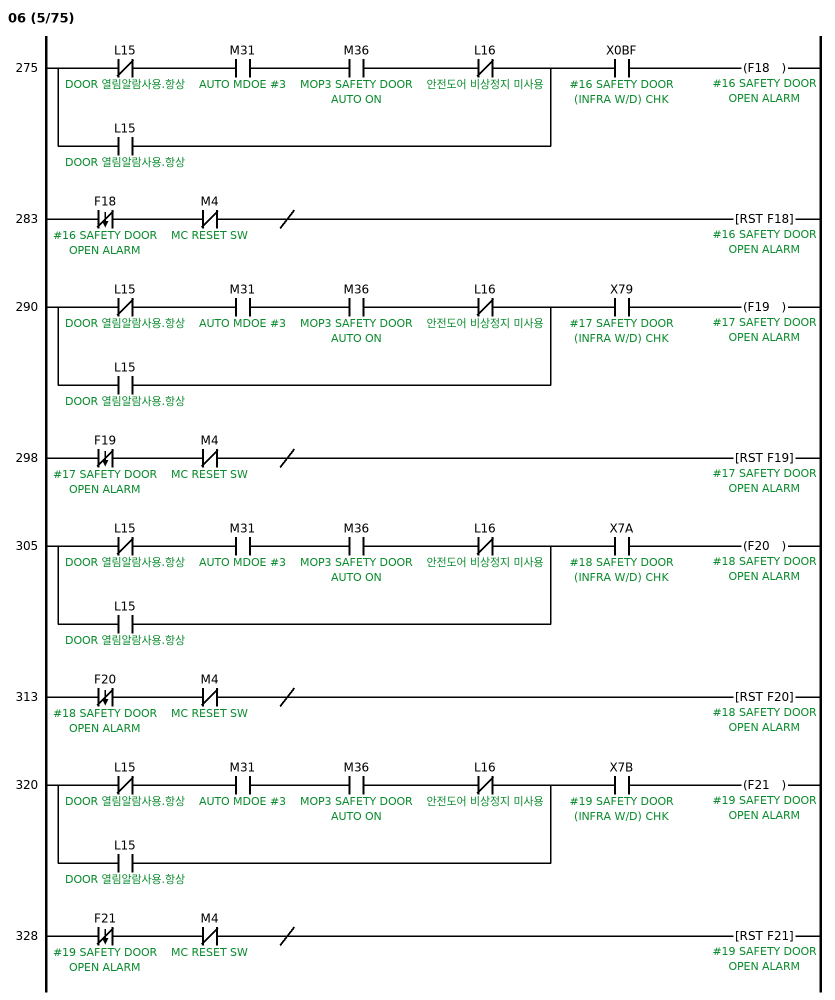
275   LDI     L15  ; DOOR 열림알람사용.항상
      AND     M31  ; AUTO MDOE #3
      AND     M36  ; MOP3 SAFETY DOOR AUTO ON
      ANI     L16  ; 안전도어 비상정지 미사용
      OR      L15  ; DOOR 열림알람사용.항상
      AND     X0BF  ; #16 SAFETY DOOR (INFRA W/D) CHK
      OUT     F18  ; #16 SAFETY DOOR OPEN ALARM
283   LDFI    F18  ; #16 SAFETY DOOR OPEN ALARM
      ANI     M4  ; MC RESET SW
      INV
      RST     F18  ; #16 SAFETY DOOR OPEN ALARM
290   LDI     L15  ; DOOR 열림알람사용.항상
      AND     M31  ; AUTO MDOE #3
      AND     M36  ; MOP3 SAFETY DOOR AUTO ON
      ANI     L16  ; 안전도어 비상정지 미사용
      OR      L15  ; DOOR 열림알람사용.항상
      AND     X79  ; #17 SAFETY DOOR (INFRA W/D) CHK
      OUT     F19  ; #17 SAFETY DOOR OPEN ALARM
298   LDFI    F19  ; #17 SAFETY DOOR OPEN ALARM
      ANI     M4  ; MC RESET SW
      INV
      RST     F19  ; #17 SAFETY DOOR OPEN ALARM
305   LDI     L15  ; DOOR 열림알람사용.항상
      AND     M31  ; AUTO MDOE #3
      AND     M36  ; MOP3 SAFETY DOOR AUTO ON
      ANI     L16  ; 안전도어 비상정지 미사용
      OR      L15  ; DOOR 열림알람사용.항상
      AND     X7A  ; #18 SAFETY DOOR (INFRA W/D) CHK
      OUT     F20  ; #18 SAFETY DOOR OPEN ALARM
313   LDFI    F20  ; #18 SAFETY DOOR OPEN ALARM
      ANI     M4  ; MC RESET SW
      INV
      RST     F20  ; #18 SAFETY DOOR OPEN ALARM
320   LDI     L15  ; DOOR 열림알람사용.항상
      AND     M31  ; AUTO MDOE #3
      AND     M36  ; MOP3 SAFETY DOOR AUTO ON
      ANI     L16  ; 안전도어 비상정지 미사용
      OR      L15  ; DOOR 열림알람사용.항상
      AND     X7B  ; #19 SAFETY DOOR (INFRA W/D) CHK
      OUT     F21  ; #19 SAFETY DOOR OPEN ALARM
328   LDFI    F21  ; #19 SAFETY DOOR OPEN ALARM
      ANI     M4  ; MC RESET SW
      INV
      RST     F21  ; #19 SAFETY DOOR OPEN ALARM
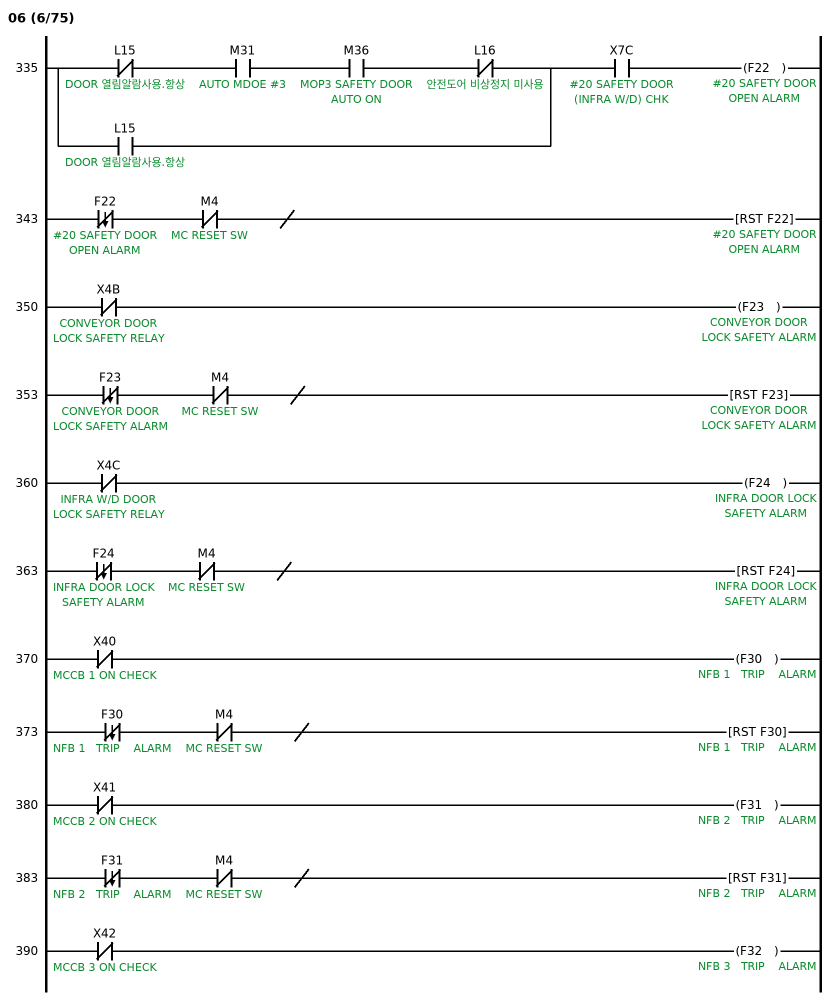
335   LDI     L15  ; DOOR 열림알람사용.항상
      AND     M31  ; AUTO MDOE #3
      AND     M36  ; MOP3 SAFETY DOOR AUTO ON
      ANI     L16  ; 안전도어 비상정지 미사용
      OR      L15  ; DOOR 열림알람사용.항상
      AND     X7C  ; #20 SAFETY DOOR (INFRA W/D) CHK
      OUT     F22  ; #20 SAFETY DOOR OPEN ALARM
343   LDFI    F22  ; #20 SAFETY DOOR OPEN ALARM
      ANI     M4  ; MC RESET SW
      INV
      RST     F22  ; #20 SAFETY DOOR OPEN ALARM
350   LDI     X4B  ; CONVEYOR DOOR LOCK SAFETY RELAY
      OUT     F23  ; CONVEYOR DOOR LOCK SAFETY ALARM
353   LDFI    F23  ; CONVEYOR DOOR LOCK SAFETY ALARM
      ANI     M4  ; MC RESET SW
      INV
      RST     F23  ; CONVEYOR DOOR LOCK SAFETY ALARM
360   LDI     X4C  ; INFRA W/D DOOR LOCK SAFETY RELAY
      OUT     F24  ; INFRA DOOR LOCK SAFETY ALARM
363   LDFI    F24  ; INFRA DOOR LOCK SAFETY ALARM
      ANI     M4  ; MC RESET SW
      INV
      RST     F24  ; INFRA DOOR LOCK SAFETY ALARM
370   LDI     X40  ; MCCB 1 ON CHECK
      OUT     F30  ; NFB 1   TRIP    ALARM
373   LDFI    F30  ; NFB 1   TRIP    ALARM
      ANI     M4  ; MC RESET SW
      INV
      RST     F30  ; NFB 1   TRIP    ALARM
380   LDI     X41  ; MCCB 2 ON CHECK
      OUT     F31  ; NFB 2   TRIP    ALARM
383   LDFI    F31  ; NFB 2   TRIP    ALARM
      ANI     M4  ; MC RESET SW
      INV
      RST     F31  ; NFB 2   TRIP    ALARM
390   LDI     X42  ; MCCB 3 ON CHECK
      OUT     F32  ; NFB 3   TRIP    ALARM
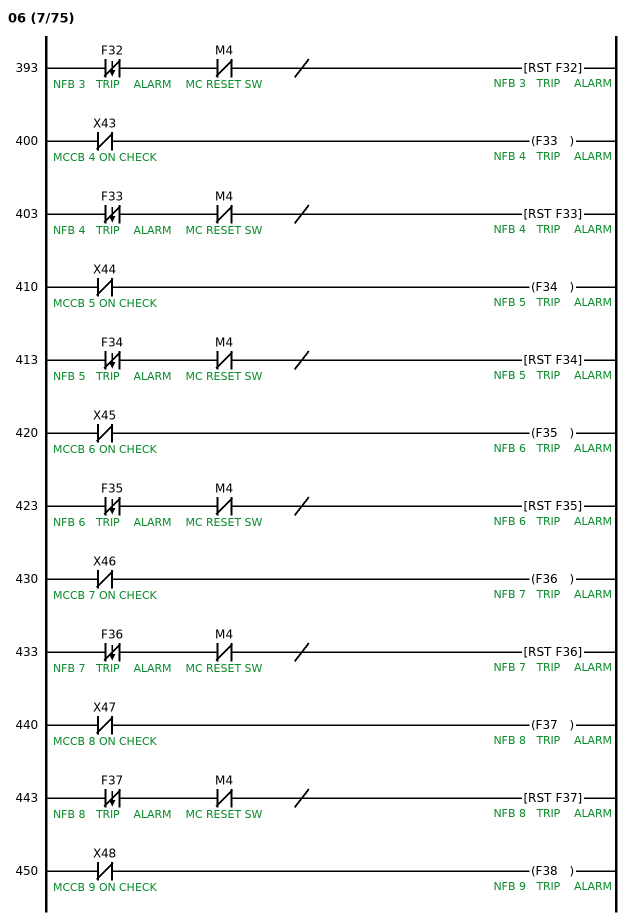
393   LDFI    F32  ; NFB 3   TRIP    ALARM
      ANI     M4  ; MC RESET SW
      INV
      RST     F32  ; NFB 3   TRIP    ALARM
400   LDI     X43  ; MCCB 4 ON CHECK
      OUT     F33  ; NFB 4   TRIP    ALARM
403   LDFI    F33  ; NFB 4   TRIP    ALARM
      ANI     M4  ; MC RESET SW
      INV
      RST     F33  ; NFB 4   TRIP    ALARM
410   LDI     X44  ; MCCB 5 ON CHECK
      OUT     F34  ; NFB 5   TRIP    ALARM
413   LDFI    F34  ; NFB 5   TRIP    ALARM
      ANI     M4  ; MC RESET SW
      INV
      RST     F34  ; NFB 5   TRIP    ALARM
420   LDI     X45  ; MCCB 6 ON CHECK
      OUT     F35  ; NFB 6   TRIP    ALARM
423   LDFI    F35  ; NFB 6   TRIP    ALARM
      ANI     M4  ; MC RESET SW
      INV
      RST     F35  ; NFB 6   TRIP    ALARM
430   LDI     X46  ; MCCB 7 ON CHECK
      OUT     F36  ; NFB 7   TRIP    ALARM
433   LDFI    F36  ; NFB 7   TRIP    ALARM
      ANI     M4  ; MC RESET SW
      INV
      RST     F36  ; NFB 7   TRIP    ALARM
440   LDI     X47  ; MCCB 8 ON CHECK
      OUT     F37  ; NFB 8   TRIP    ALARM
443   LDFI    F37  ; NFB 8   TRIP    ALARM
      ANI     M4  ; MC RESET SW
      INV
      RST     F37  ; NFB 8   TRIP    ALARM
450   LDI     X48  ; MCCB 9 ON CHECK
      OUT     F38  ; NFB 9   TRIP    ALARM
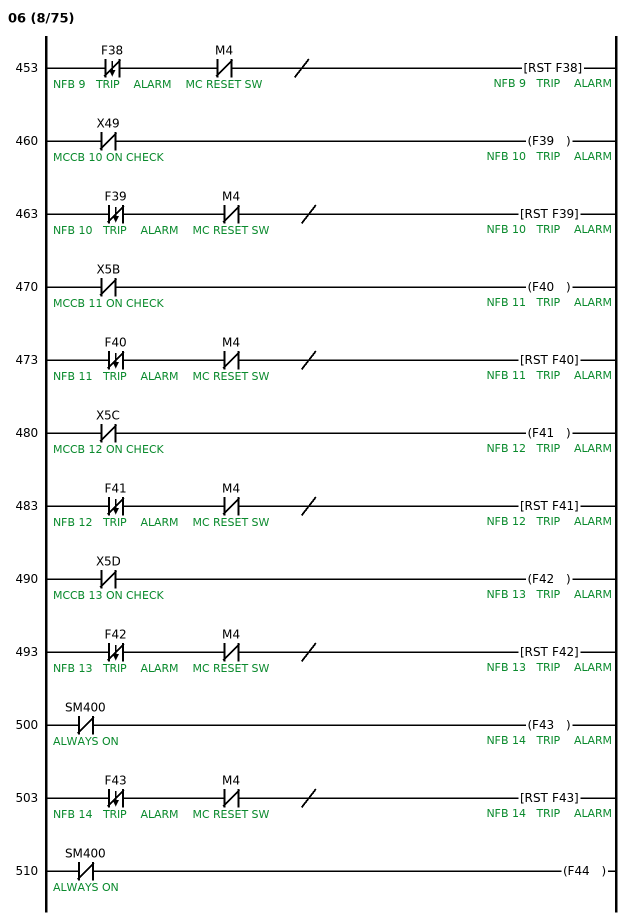
453   LDFI    F38  ; NFB 9   TRIP    ALARM
      ANI     M4  ; MC RESET SW
      INV
      RST     F38  ; NFB 9   TRIP    ALARM
460   LDI     X49  ; MCCB 10 ON CHECK
      OUT     F39  ; NFB 10   TRIP    ALARM
463   LDFI    F39  ; NFB 10   TRIP    ALARM
      ANI     M4  ; MC RESET SW
      INV
      RST     F39  ; NFB 10   TRIP    ALARM
470   LDI     X5B  ; MCCB 11 ON CHECK
      OUT     F40  ; NFB 11   TRIP    ALARM
473   LDFI    F40  ; NFB 11   TRIP    ALARM
      ANI     M4  ; MC RESET SW
      INV
      RST     F40  ; NFB 11   TRIP    ALARM
480   LDI     X5C  ; MCCB 12 ON CHECK
      OUT     F41  ; NFB 12   TRIP    ALARM
483   LDFI    F41  ; NFB 12   TRIP    ALARM
      ANI     M4  ; MC RESET SW
      INV
      RST     F41  ; NFB 12   TRIP    ALARM
490   LDI     X5D  ; MCCB 13 ON CHECK
      OUT     F42  ; NFB 13   TRIP    ALARM
493   LDFI    F42  ; NFB 13   TRIP    ALARM
      ANI     M4  ; MC RESET SW
      INV
      RST     F42  ; NFB 13   TRIP    ALARM
500   LDI     SM400  ; ALWAYS ON
      OUT     F43  ; NFB 14   TRIP    ALARM
503   LDFI    F43  ; NFB 14   TRIP    ALARM
      ANI     M4  ; MC RESET SW
      INV
      RST     F43  ; NFB 14   TRIP    ALARM
510   LDI     SM400  ; ALWAYS ON
      OUT     F44
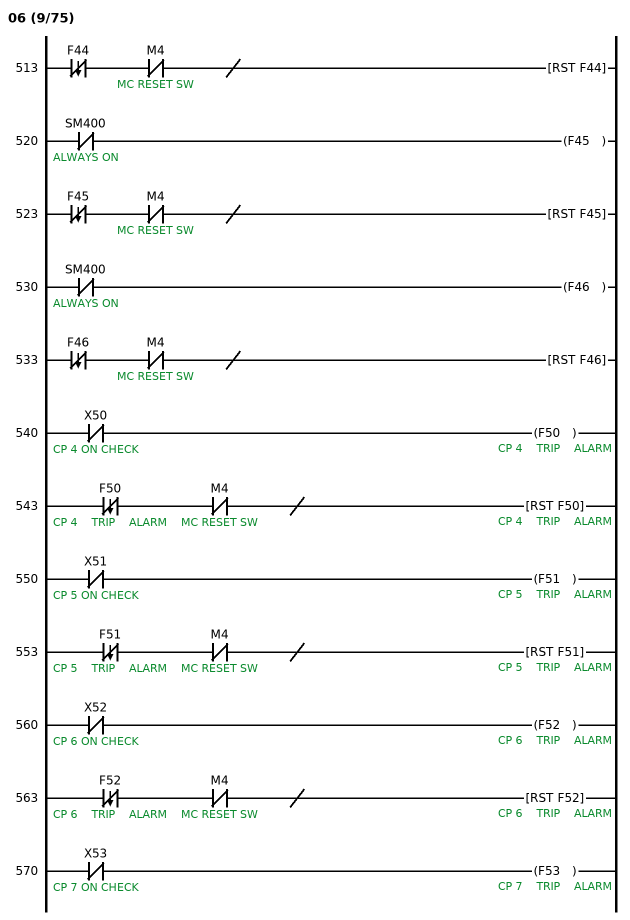
513   LDFI    F44
      ANI     M4  ; MC RESET SW
      INV
      RST     F44
520   LDI     SM400  ; ALWAYS ON
      OUT     F45
523   LDFI    F45
      ANI     M4  ; MC RESET SW
      INV
      RST     F45
530   LDI     SM400  ; ALWAYS ON
      OUT     F46
533   LDFI    F46
      ANI     M4  ; MC RESET SW
      INV
      RST     F46
540   LDI     X50  ; CP 4 ON CHECK
      OUT     F50  ; CP 4    TRIP    ALARM
543   LDFI    F50  ; CP 4    TRIP    ALARM
      ANI     M4  ; MC RESET SW
      INV
      RST     F50  ; CP 4    TRIP    ALARM
550   LDI     X51  ; CP 5 ON CHECK
      OUT     F51  ; CP 5    TRIP    ALARM
553   LDFI    F51  ; CP 5    TRIP    ALARM
      ANI     M4  ; MC RESET SW
      INV
      RST     F51  ; CP 5    TRIP    ALARM
560   LDI     X52  ; CP 6 ON CHECK
      OUT     F52  ; CP 6    TRIP    ALARM
563   LDFI    F52  ; CP 6    TRIP    ALARM
      ANI     M4  ; MC RESET SW
      INV
      RST     F52  ; CP 6    TRIP    ALARM
570   LDI     X53  ; CP 7 ON CHECK
      OUT     F53  ; CP 7    TRIP    ALARM
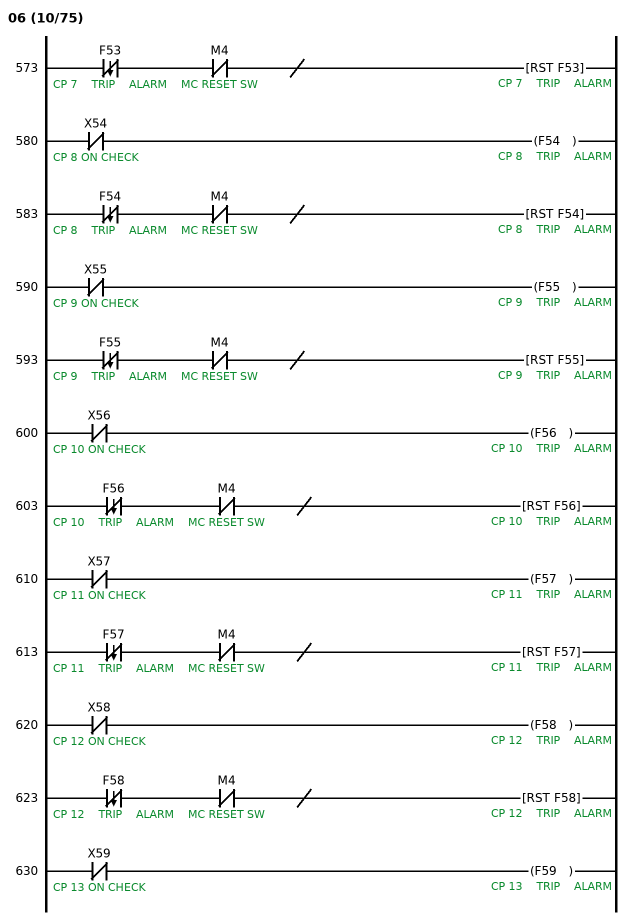
573   LDFI    F53  ; CP 7    TRIP    ALARM
      ANI     M4  ; MC RESET SW
      INV
      RST     F53  ; CP 7    TRIP    ALARM
580   LDI     X54  ; CP 8 ON CHECK
      OUT     F54  ; CP 8    TRIP    ALARM
583   LDFI    F54  ; CP 8    TRIP    ALARM
      ANI     M4  ; MC RESET SW
      INV
      RST     F54  ; CP 8    TRIP    ALARM
590   LDI     X55  ; CP 9 ON CHECK
      OUT     F55  ; CP 9    TRIP    ALARM
593   LDFI    F55  ; CP 9    TRIP    ALARM
      ANI     M4  ; MC RESET SW
      INV
      RST     F55  ; CP 9    TRIP    ALARM
600   LDI     X56  ; CP 10 ON CHECK
      OUT     F56  ; CP 10    TRIP    ALARM
603   LDFI    F56  ; CP 10    TRIP    ALARM
      ANI     M4  ; MC RESET SW
      INV
      RST     F56  ; CP 10    TRIP    ALARM
610   LDI     X57  ; CP 11 ON CHECK
      OUT     F57  ; CP 11    TRIP    ALARM
613   LDFI    F57  ; CP 11    TRIP    ALARM
      ANI     M4  ; MC RESET SW
      INV
      RST     F57  ; CP 11    TRIP    ALARM
620   LDI     X58  ; CP 12 ON CHECK
      OUT     F58  ; CP 12    TRIP    ALARM
623   LDFI    F58  ; CP 12    TRIP    ALARM
      ANI     M4  ; MC RESET SW
      INV
      RST     F58  ; CP 12    TRIP    ALARM
630   LDI     X59  ; CP 13 ON CHECK
      OUT     F59  ; CP 13    TRIP    ALARM
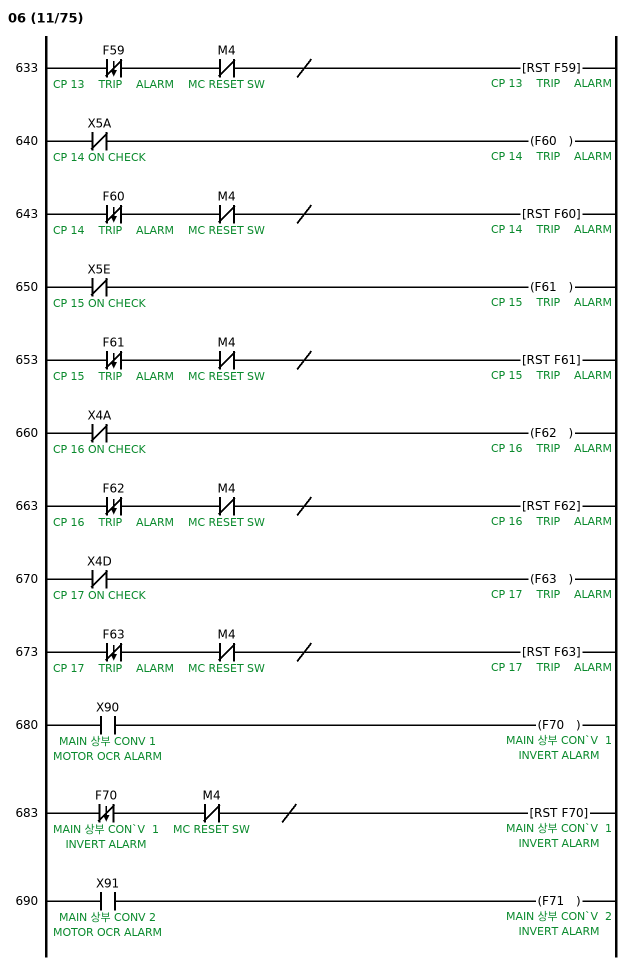
633   LDFI    F59  ; CP 13    TRIP    ALARM
      ANI     M4  ; MC RESET SW
      INV
      RST     F59  ; CP 13    TRIP    ALARM
640   LDI     X5A  ; CP 14 ON CHECK
      OUT     F60  ; CP 14    TRIP    ALARM
643   LDFI    F60  ; CP 14    TRIP    ALARM
      ANI     M4  ; MC RESET SW
      INV
      RST     F60  ; CP 14    TRIP    ALARM
650   LDI     X5E  ; CP 15 ON CHECK
      OUT     F61  ; CP 15    TRIP    ALARM
653   LDFI    F61  ; CP 15    TRIP    ALARM
      ANI     M4  ; MC RESET SW
      INV
      RST     F61  ; CP 15    TRIP    ALARM
660   LDI     X4A  ; CP 16 ON CHECK
      OUT     F62  ; CP 16    TRIP    ALARM
663   LDFI    F62  ; CP 16    TRIP    ALARM
      ANI     M4  ; MC RESET SW
      INV
      RST     F62  ; CP 16    TRIP    ALARM
670   LDI     X4D  ; CP 17 ON CHECK
      OUT     F63  ; CP 17    TRIP    ALARM
673   LDFI    F63  ; CP 17    TRIP    ALARM
      ANI     M4  ; MC RESET SW
      INV
      RST     F63  ; CP 17    TRIP    ALARM
680   LD      X90  ; MAIN 상부 CONV 1 MOTOR OCR ALARM
      OUT     F70  ; MAIN 상부 CON`V  1 INVERT ALARM
683   LDFI    F70  ; MAIN 상부 CON`V  1 INVERT ALARM
      ANI     M4  ; MC RESET SW
      INV
      RST     F70  ; MAIN 상부 CON`V  1 INVERT ALARM
690   LD      X91  ; MAIN 상부 CONV 2 MOTOR OCR ALARM
      OUT     F71  ; MAIN 상부 CON`V  2 INVERT ALARM
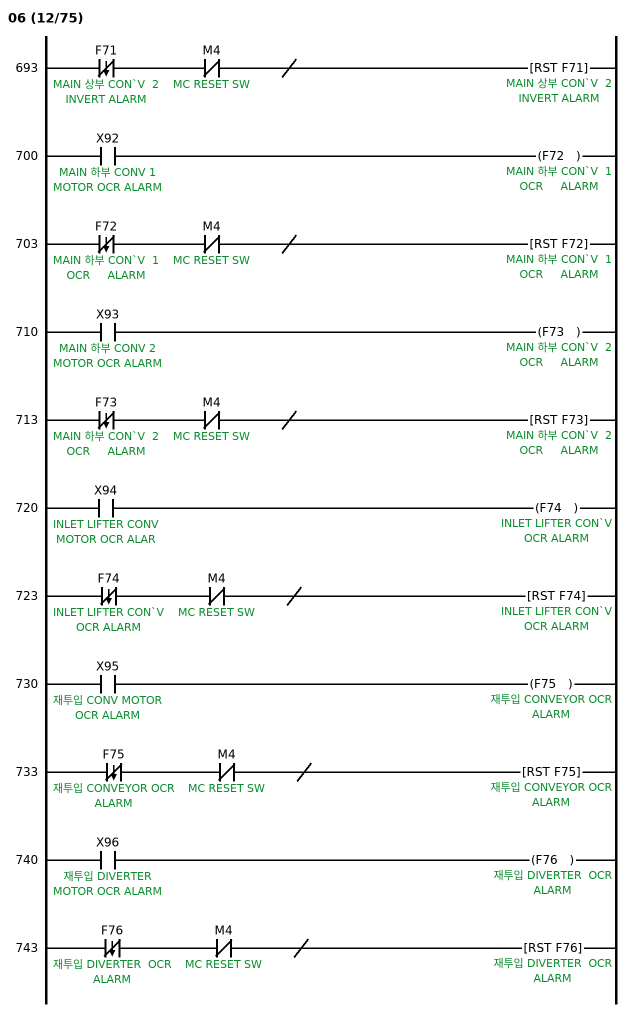
693   LDFI    F71  ; MAIN 상부 CON`V  2 INVERT ALARM
      ANI     M4  ; MC RESET SW
      INV
      RST     F71  ; MAIN 상부 CON`V  2 INVERT ALARM
700   LD      X92  ; MAIN 하부 CONV 1 MOTOR OCR ALARM
      OUT     F72  ; MAIN 하부 CON`V  1 OCR     ALARM
703   LDFI    F72  ; MAIN 하부 CON`V  1 OCR     ALARM
      ANI     M4  ; MC RESET SW
      INV
      RST     F72  ; MAIN 하부 CON`V  1 OCR     ALARM
710   LD      X93  ; MAIN 하부 CONV 2 MOTOR OCR ALARM
      OUT     F73  ; MAIN 하부 CON`V  2 OCR     ALARM
713   LDFI    F73  ; MAIN 하부 CON`V  2 OCR     ALARM
      ANI     M4  ; MC RESET SW
      INV
      RST     F73  ; MAIN 하부 CON`V  2 OCR     ALARM
720   LD      X94  ; INLET LIFTER CONV MOTOR OCR ALAR
      OUT     F74  ; INLET LIFTER CON`V OCR ALARM
723   LDFI    F74  ; INLET LIFTER CON`V OCR ALARM
      ANI     M4  ; MC RESET SW
      INV
      RST     F74  ; INLET LIFTER CON`V OCR ALARM
730   LD      X95  ; 재투입 CONV MOTOR OCR ALARM
      OUT     F75  ; 재투입 CONVEYOR OCR     ALARM
733   LDFI    F75  ; 재투입 CONVEYOR OCR     ALARM
      ANI     M4  ; MC RESET SW
      INV
      RST     F75  ; 재투입 CONVEYOR OCR     ALARM
740   LD      X96  ; 재투입 DIVERTER MOTOR OCR ALARM
      OUT     F76  ; 재투입 DIVERTER  OCR     ALARM
743   LDFI    F76  ; 재투입 DIVERTER  OCR     ALARM
      ANI     M4  ; MC RESET SW
      INV
      RST     F76  ; 재투입 DIVERTER  OCR     ALARM
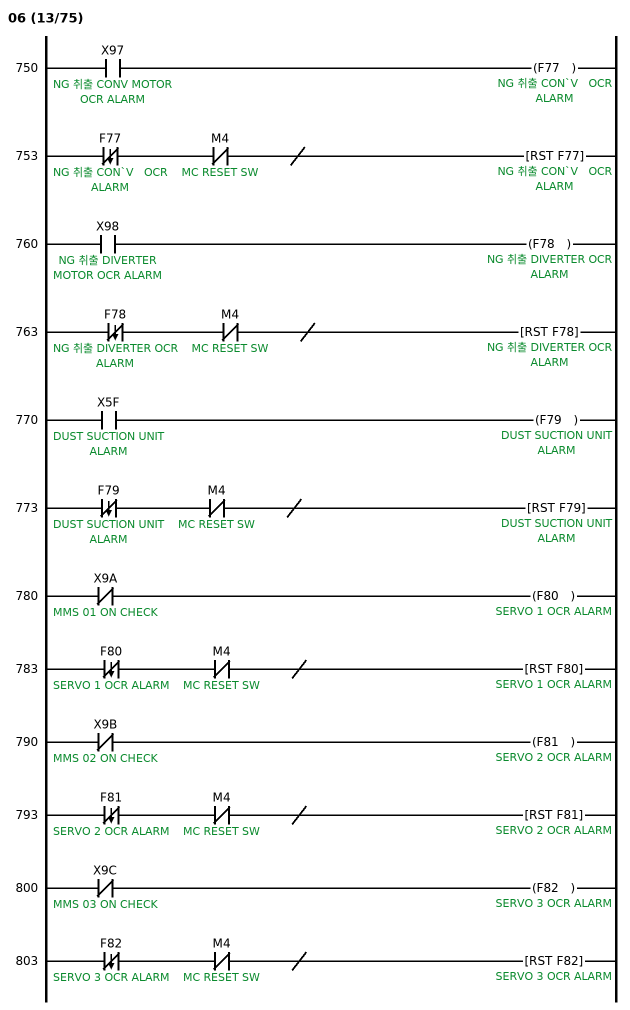
750   LD      X97  ; NG 취출 CONV MOTOR OCR ALARM
      OUT     F77  ; NG 취출 CON`V   OCR     ALARM
753   LDFI    F77  ; NG 취출 CON`V   OCR     ALARM
      ANI     M4  ; MC RESET SW
      INV
      RST     F77  ; NG 취출 CON`V   OCR     ALARM
760   LD      X98  ; NG 취출 DIVERTER MOTOR OCR ALARM
      OUT     F78  ; NG 취출 DIVERTER OCR ALARM
763   LDFI    F78  ; NG 취출 DIVERTER OCR ALARM
      ANI     M4  ; MC RESET SW
      INV
      RST     F78  ; NG 취출 DIVERTER OCR ALARM
770   LD      X5F  ; DUST SUCTION UNIT ALARM
      OUT     F79  ; DUST SUCTION UNIT ALARM
773   LDFI    F79  ; DUST SUCTION UNIT ALARM
      ANI     M4  ; MC RESET SW
      INV
      RST     F79  ; DUST SUCTION UNIT ALARM
780   LDI     X9A  ; MMS 01 ON CHECK
      OUT     F80  ; SERVO 1 OCR ALARM
783   LDFI    F80  ; SERVO 1 OCR ALARM
      ANI     M4  ; MC RESET SW
      INV
      RST     F80  ; SERVO 1 OCR ALARM
790   LDI     X9B  ; MMS 02 ON CHECK
      OUT     F81  ; SERVO 2 OCR ALARM
793   LDFI    F81  ; SERVO 2 OCR ALARM
      ANI     M4  ; MC RESET SW
      INV
      RST     F81  ; SERVO 2 OCR ALARM
800   LDI     X9C  ; MMS 03 ON CHECK
      OUT     F82  ; SERVO 3 OCR ALARM
803   LDFI    F82  ; SERVO 3 OCR ALARM
      ANI     M4  ; MC RESET SW
      INV
      RST     F82  ; SERVO 3 OCR ALARM
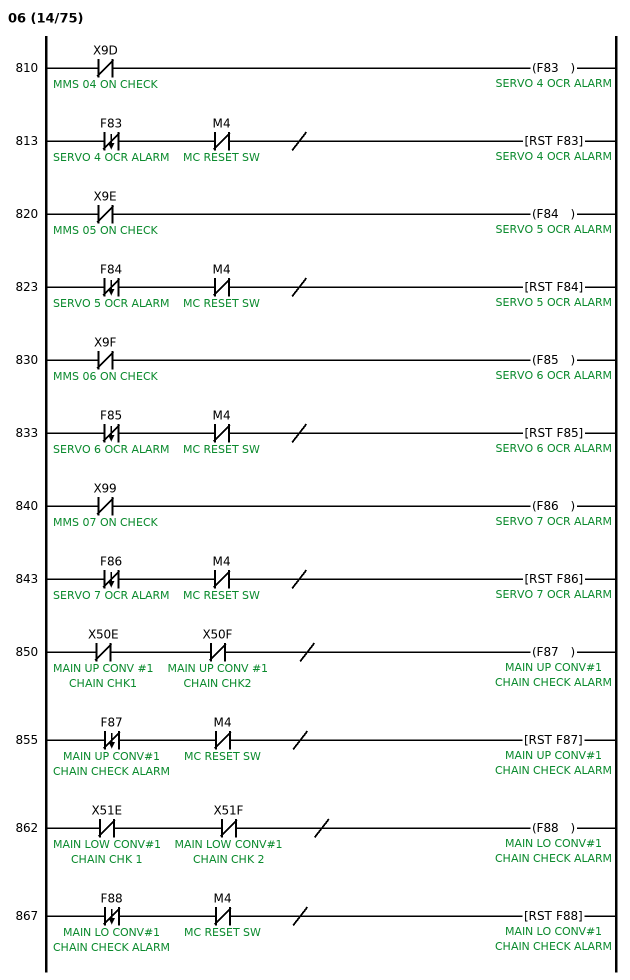
810   LDI     X9D  ; MMS 04 ON CHECK
      OUT     F83  ; SERVO 4 OCR ALARM
813   LDFI    F83  ; SERVO 4 OCR ALARM
      ANI     M4  ; MC RESET SW
      INV
      RST     F83  ; SERVO 4 OCR ALARM
820   LDI     X9E  ; MMS 05 ON CHECK
      OUT     F84  ; SERVO 5 OCR ALARM
823   LDFI    F84  ; SERVO 5 OCR ALARM
      ANI     M4  ; MC RESET SW
      INV
      RST     F84  ; SERVO 5 OCR ALARM
830   LDI     X9F  ; MMS 06 ON CHECK
      OUT     F85  ; SERVO 6 OCR ALARM
833   LDFI    F85  ; SERVO 6 OCR ALARM
      ANI     M4  ; MC RESET SW
      INV
      RST     F85  ; SERVO 6 OCR ALARM
840   LDI     X99  ; MMS 07 ON CHECK
      OUT     F86  ; SERVO 7 OCR ALARM
843   LDFI    F86  ; SERVO 7 OCR ALARM
      ANI     M4  ; MC RESET SW
      INV
      RST     F86  ; SERVO 7 OCR ALARM
850   LDI     X50E  ; MAIN UP CONV #1 CHAIN CHK1
      ANI     X50F  ; MAIN UP CONV #1 CHAIN CHK2
      INV
      OUT     F87  ; MAIN UP CONV#1 CHAIN CHECK ALARM
855   LDFI    F87  ; MAIN UP CONV#1 CHAIN CHECK ALARM
      ANI     M4  ; MC RESET SW
      INV
      RST     F87  ; MAIN UP CONV#1 CHAIN CHECK ALARM
862   LDI     X51E  ; MAIN LOW CONV#1 CHAIN CHK 1
      ANI     X51F  ; MAIN LOW CONV#1 CHAIN CHK 2
      INV
      OUT     F88  ; MAIN LO CONV#1 CHAIN CHECK ALARM
867   LDFI    F88  ; MAIN LO CONV#1 CHAIN CHECK ALARM
      ANI     M4  ; MC RESET SW
      INV
      RST     F88  ; MAIN LO CONV#1 CHAIN CHECK ALARM
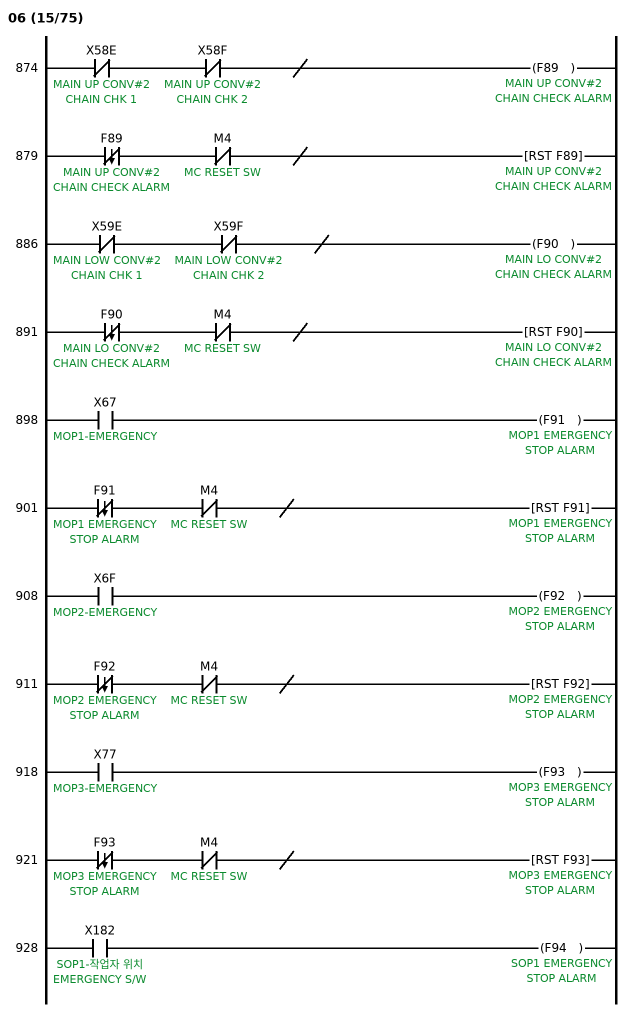
874   LDI     X58E  ; MAIN UP CONV#2 CHAIN CHK 1
      ANI     X58F  ; MAIN UP CONV#2 CHAIN CHK 2
      INV
      OUT     F89  ; MAIN UP CONV#2 CHAIN CHECK ALARM
879   LDFI    F89  ; MAIN UP CONV#2 CHAIN CHECK ALARM
      ANI     M4  ; MC RESET SW
      INV
      RST     F89  ; MAIN UP CONV#2 CHAIN CHECK ALARM
886   LDI     X59E  ; MAIN LOW CONV#2 CHAIN CHK 1
      ANI     X59F  ; MAIN LOW CONV#2 CHAIN CHK 2
      INV
      OUT     F90  ; MAIN LO CONV#2 CHAIN CHECK ALARM
891   LDFI    F90  ; MAIN LO CONV#2 CHAIN CHECK ALARM
      ANI     M4  ; MC RESET SW
      INV
      RST     F90  ; MAIN LO CONV#2 CHAIN CHECK ALARM
898   LD      X67  ; MOP1-EMERGENCY
      OUT     F91  ; MOP1 EMERGENCY STOP ALARM
901   LDFI    F91  ; MOP1 EMERGENCY STOP ALARM
      ANI     M4  ; MC RESET SW
      INV
      RST     F91  ; MOP1 EMERGENCY STOP ALARM
908   LD      X6F  ; MOP2-EMERGENCY
      OUT     F92  ; MOP2 EMERGENCY STOP ALARM
911   LDFI    F92  ; MOP2 EMERGENCY STOP ALARM
      ANI     M4  ; MC RESET SW
      INV
      RST     F92  ; MOP2 EMERGENCY STOP ALARM
918   LD      X77  ; MOP3-EMERGENCY
      OUT     F93  ; MOP3 EMERGENCY STOP ALARM
921   LDFI    F93  ; MOP3 EMERGENCY STOP ALARM
      ANI     M4  ; MC RESET SW
      INV
      RST     F93  ; MOP3 EMERGENCY STOP ALARM
928   LD      X182  ; SOP1-작업자 위치 EMERGENCY S/W
      OUT     F94  ; SOP1 EMERGENCY STOP ALARM
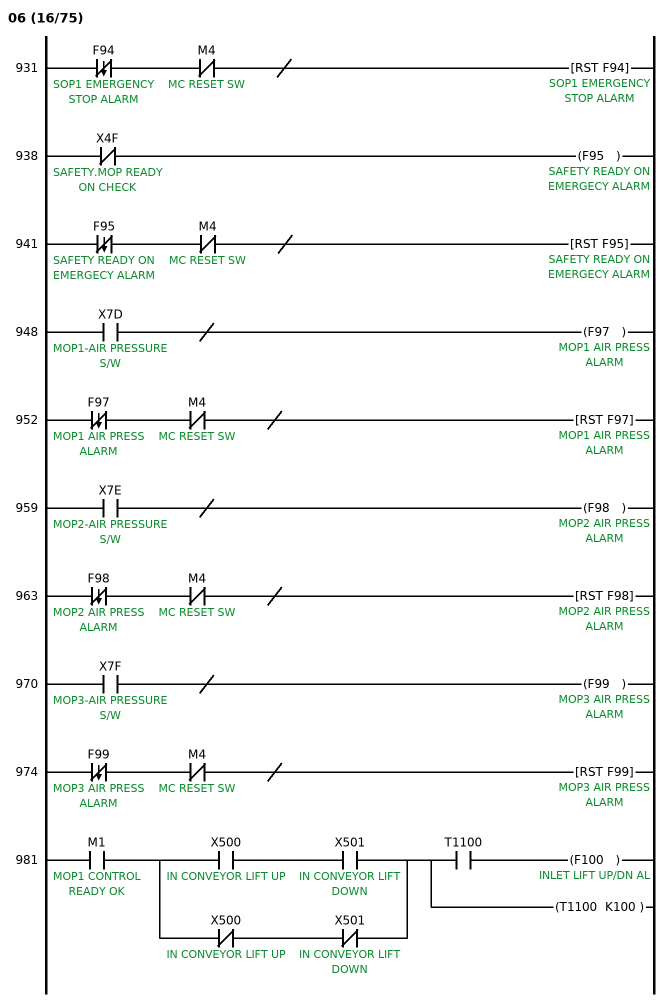
931   LDFI    F94  ; SOP1 EMERGENCY STOP ALARM
      ANI     M4  ; MC RESET SW
      INV
      RST     F94  ; SOP1 EMERGENCY STOP ALARM
938   LDI     X4F  ; SAFETY.MOP READY ON CHECK
      OUT     F95  ; SAFETY READY ON EMERGECY ALARM
941   LDFI    F95  ; SAFETY READY ON EMERGECY ALARM
      ANI     M4  ; MC RESET SW
      INV
      RST     F95  ; SAFETY READY ON EMERGECY ALARM
948   LD      X7D  ; MOP1-AIR PRESSURE S/W
      INV
      OUT     F97  ; MOP1 AIR PRESS ALARM
952   LDFI    F97  ; MOP1 AIR PRESS ALARM
      ANI     M4  ; MC RESET SW
      INV
      RST     F97  ; MOP1 AIR PRESS ALARM
959   LD      X7E  ; MOP2-AIR PRESSURE S/W
      INV
      OUT     F98  ; MOP2 AIR PRESS ALARM
963   LDFI    F98  ; MOP2 AIR PRESS ALARM
      ANI     M4  ; MC RESET SW
      INV
      RST     F98  ; MOP2 AIR PRESS ALARM
970   LD      X7F  ; MOP3-AIR PRESSURE S/W
      INV
      OUT     F99  ; MOP3 AIR PRESS ALARM
974   LDFI    F99  ; MOP3 AIR PRESS ALARM
      ANI     M4  ; MC RESET SW
      INV
      RST     F99  ; MOP3 AIR PRESS ALARM
981   LD      M1  ; MOP1 CONTROL READY OK
      LD      X500  ; IN CONVEYOR LIFT UP
      AND     X501  ; IN CONVEYOR LIFT DOWN
      LDI     X500  ; IN CONVEYOR LIFT UP
      ANI     X501  ; IN CONVEYOR LIFT DOWN
      ORB
      ANB
      MPS
      AND     T1100
      OUT     F100  ; INLET LIFT UP/DN AL
      MPP
      OUT     T1100 K100
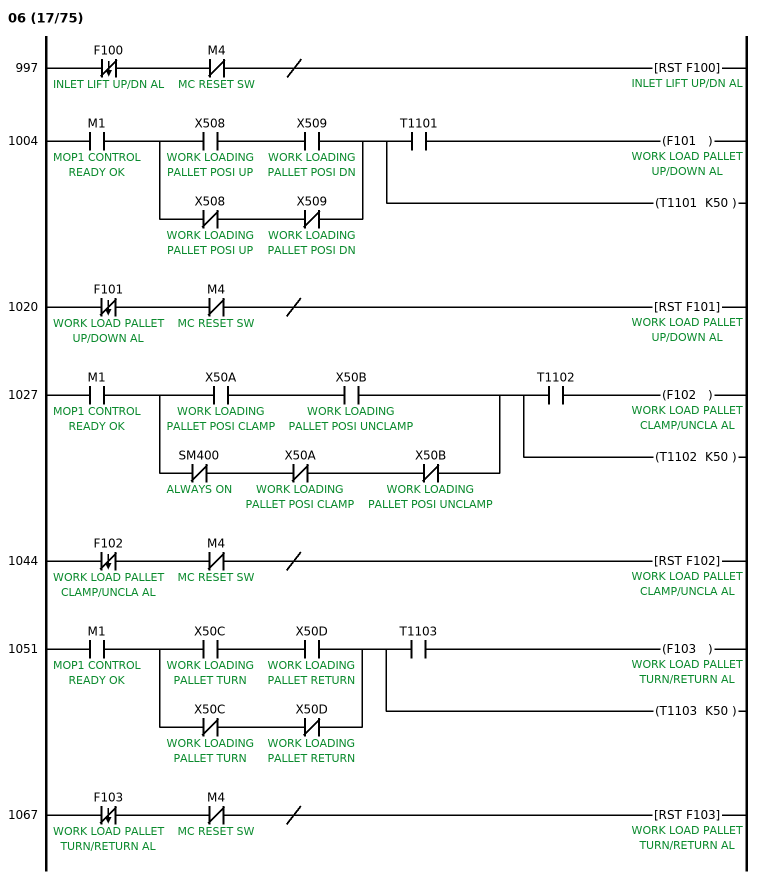
997   LDFI    F100  ; INLET LIFT UP/DN AL
      ANI     M4  ; MC RESET SW
      INV
      RST     F100  ; INLET LIFT UP/DN AL
1004  LD      M1  ; MOP1 CONTROL READY OK
      LD      X508  ; WORK LOADING PALLET POSI UP
      AND     X509  ; WORK LOADING PALLET POSI DN
      LDI     X508  ; WORK LOADING PALLET POSI UP
      ANI     X509  ; WORK LOADING PALLET POSI DN
      ORB
      ANB
      MPS
      AND     T1101
      OUT     F101  ; WORK LOAD PALLET UP/DOWN AL
      MPP
      OUT     T1101 K50
1020  LDFI    F101  ; WORK LOAD PALLET UP/DOWN AL
      ANI     M4  ; MC RESET SW
      INV
      RST     F101  ; WORK LOAD PALLET UP/DOWN AL
1027  LD      M1  ; MOP1 CONTROL READY OK
      LD      X50A  ; WORK LOADING PALLET POSI CLAMP
      AND     X50B  ; WORK LOADING PALLET POSI UNCLAMP
      LDI     SM400  ; ALWAYS ON
      ANI     X50A  ; WORK LOADING PALLET POSI CLAMP
      ANI     X50B  ; WORK LOADING PALLET POSI UNCLAMP
      ORB
      ANB
      MPS
      AND     T1102
      OUT     F102  ; WORK LOAD PALLET CLAMP/UNCLA AL
      MPP
      OUT     T1102 K50
1044  LDFI    F102  ; WORK LOAD PALLET CLAMP/UNCLA AL
      ANI     M4  ; MC RESET SW
      INV
      RST     F102  ; WORK LOAD PALLET CLAMP/UNCLA AL
1051  LD      M1  ; MOP1 CONTROL READY OK
      LD      X50C  ; WORK LOADING PALLET TURN
      AND     X50D  ; WORK LOADING PALLET RETURN
      LDI     X50C  ; WORK LOADING PALLET TURN
      ANI     X50D  ; WORK LOADING PALLET RETURN
      ORB
      ANB
      MPS
      AND     T1103
      OUT     F103  ; WORK LOAD PALLET TURN/RETURN AL
      MPP
      OUT     T1103 K50
1067  LDFI    F103  ; WORK LOAD PALLET TURN/RETURN AL
      ANI     M4  ; MC RESET SW
      INV
      RST     F103  ; WORK LOAD PALLET TURN/RETURN AL
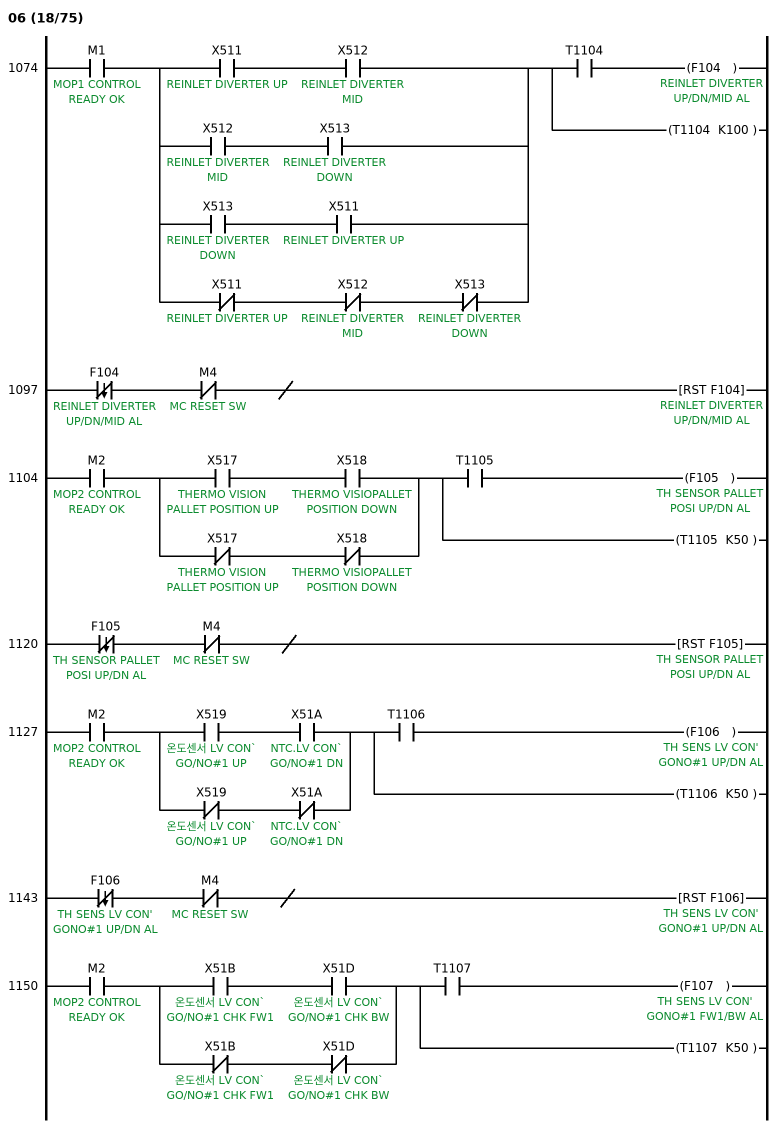
1074  LD      M1  ; MOP1 CONTROL READY OK
      LD      X511  ; REINLET DIVERTER UP
      AND     X512  ; REINLET DIVERTER MID
      LD      X512  ; REINLET DIVERTER MID
      AND     X513  ; REINLET DIVERTER DOWN
      ORB
      LD      X513  ; REINLET DIVERTER DOWN
      AND     X511  ; REINLET DIVERTER UP
      ORB
      LDI     X511  ; REINLET DIVERTER UP
      ANI     X512  ; REINLET DIVERTER MID
      ANI     X513  ; REINLET DIVERTER DOWN
      ORB
      ANB
      MPS
      AND     T1104
      OUT     F104  ; REINLET DIVERTER UP/DN/MID AL
      MPP
      OUT     T1104 K100
1097  LDFI    F104  ; REINLET DIVERTER UP/DN/MID AL
      ANI     M4  ; MC RESET SW
      INV
      RST     F104  ; REINLET DIVERTER UP/DN/MID AL
1104  LD      M2  ; MOP2 CONTROL READY OK
      LD      X517  ; THERMO VISION PALLET POSITION UP
      AND     X518  ; THERMO VISIOPALLET POSITION DOWN
      LDI     X517  ; THERMO VISION PALLET POSITION UP
      ANI     X518  ; THERMO VISIOPALLET POSITION DOWN
      ORB
      ANB
      MPS
      AND     T1105
      OUT     F105  ; TH SENSOR PALLET POSI UP/DN AL
      MPP
      OUT     T1105 K50
1120  LDFI    F105  ; TH SENSOR PALLET POSI UP/DN AL
      ANI     M4  ; MC RESET SW
      INV
      RST     F105  ; TH SENSOR PALLET POSI UP/DN AL
1127  LD      M2  ; MOP2 CONTROL READY OK
      LD      X519  ; 온도센서 LV CON` GO/NO#1 UP
      AND     X51A  ; NTC.LV CON` GO/NO#1 DN
      LDI     X519  ; 온도센서 LV CON` GO/NO#1 UP
      ANI     X51A  ; NTC.LV CON` GO/NO#1 DN
      ORB
      ANB
      MPS
      AND     T1106
      OUT     F106  ; TH SENS LV CON' GONO#1 UP/DN AL
      MPP
      OUT     T1106 K50
1143  LDFI    F106  ; TH SENS LV CON' GONO#1 UP/DN AL
      ANI     M4  ; MC RESET SW
      INV
      RST     F106  ; TH SENS LV CON' GONO#1 UP/DN AL
1150  LD      M2  ; MOP2 CONTROL READY OK
      LD      X51B  ; 온도센서 LV CON` GO/NO#1 CHK FW1
      AND     X51D  ; 온도센서 LV CON` GO/NO#1 CHK BW
      LDI     X51B  ; 온도센서 LV CON` GO/NO#1 CHK FW1
      ANI     X51D  ; 온도센서 LV CON` GO/NO#1 CHK BW
      ORB
      ANB
      MPS
      AND     T1107
      OUT     F107  ; TH SENS LV CON' GONO#1 FW1/BW AL
      MPP
      OUT     T1107 K50
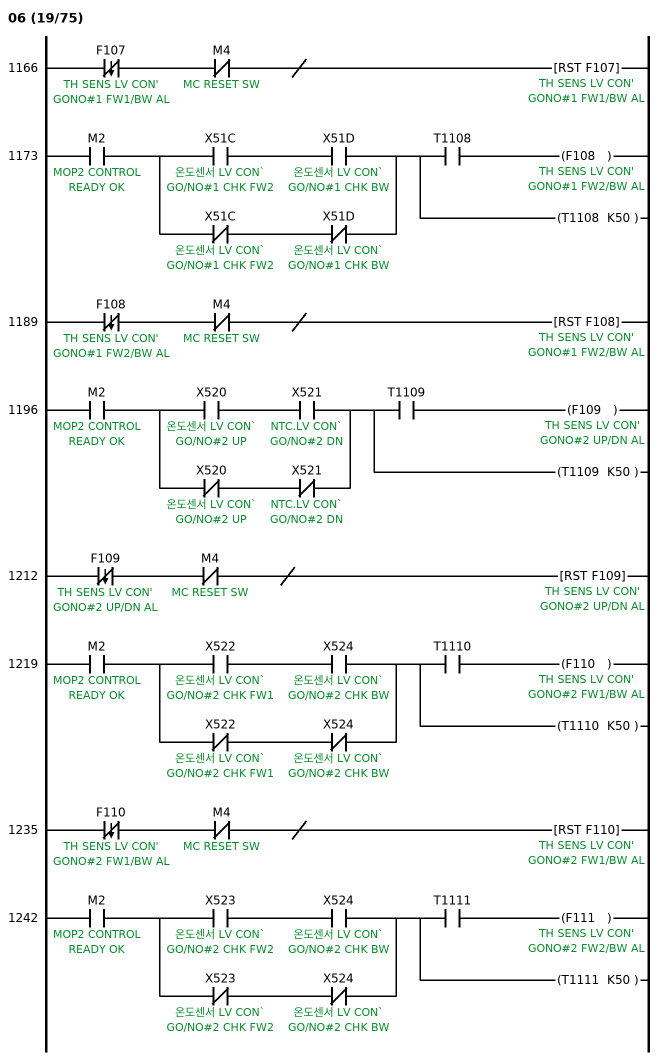
1166  LDFI    F107  ; TH SENS LV CON' GONO#1 FW1/BW AL
      ANI     M4  ; MC RESET SW
      INV
      RST     F107  ; TH SENS LV CON' GONO#1 FW1/BW AL
1173  LD      M2  ; MOP2 CONTROL READY OK
      LD      X51C  ; 온도센서 LV CON` GO/NO#1 CHK FW2
      AND     X51D  ; 온도센서 LV CON` GO/NO#1 CHK BW
      LDI     X51C  ; 온도센서 LV CON` GO/NO#1 CHK FW2
      ANI     X51D  ; 온도센서 LV CON` GO/NO#1 CHK BW
      ORB
      ANB
      MPS
      AND     T1108
      OUT     F108  ; TH SENS LV CON' GONO#1 FW2/BW AL
      MPP
      OUT     T1108 K50
1189  LDFI    F108  ; TH SENS LV CON' GONO#1 FW2/BW AL
      ANI     M4  ; MC RESET SW
      INV
      RST     F108  ; TH SENS LV CON' GONO#1 FW2/BW AL
1196  LD      M2  ; MOP2 CONTROL READY OK
      LD      X520  ; 온도센서 LV CON` GO/NO#2 UP
      AND     X521  ; NTC.LV CON` GO/NO#2 DN
      LDI     X520  ; 온도센서 LV CON` GO/NO#2 UP
      ANI     X521  ; NTC.LV CON` GO/NO#2 DN
      ORB
      ANB
      MPS
      AND     T1109
      OUT     F109  ; TH SENS LV CON' GONO#2 UP/DN AL
      MPP
      OUT     T1109 K50
1212  LDFI    F109  ; TH SENS LV CON' GONO#2 UP/DN AL
      ANI     M4  ; MC RESET SW
      INV
      RST     F109  ; TH SENS LV CON' GONO#2 UP/DN AL
1219  LD      M2  ; MOP2 CONTROL READY OK
      LD      X522  ; 온도센서 LV CON` GO/NO#2 CHK FW1
      AND     X524  ; 온도센서 LV CON` GO/NO#2 CHK BW
      LDI     X522  ; 온도센서 LV CON` GO/NO#2 CHK FW1
      ANI     X524  ; 온도센서 LV CON` GO/NO#2 CHK BW
      ORB
      ANB
      MPS
      AND     T1110
      OUT     F110  ; TH SENS LV CON' GONO#2 FW1/BW AL
      MPP
      OUT     T1110 K50
1235  LDFI    F110  ; TH SENS LV CON' GONO#2 FW1/BW AL
      ANI     M4  ; MC RESET SW
      INV
      RST     F110  ; TH SENS LV CON' GONO#2 FW1/BW AL
1242  LD      M2  ; MOP2 CONTROL READY OK
      LD      X523  ; 온도센서 LV CON` GO/NO#2 CHK FW2
      AND     X524  ; 온도센서 LV CON` GO/NO#2 CHK BW
      LDI     X523  ; 온도센서 LV CON` GO/NO#2 CHK FW2
      ANI     X524  ; 온도센서 LV CON` GO/NO#2 CHK BW
      ORB
      ANB
      MPS
      AND     T1111
      OUT     F111  ; TH SENS LV CON' GONO#2 FW2/BW AL
      MPP
      OUT     T1111 K50
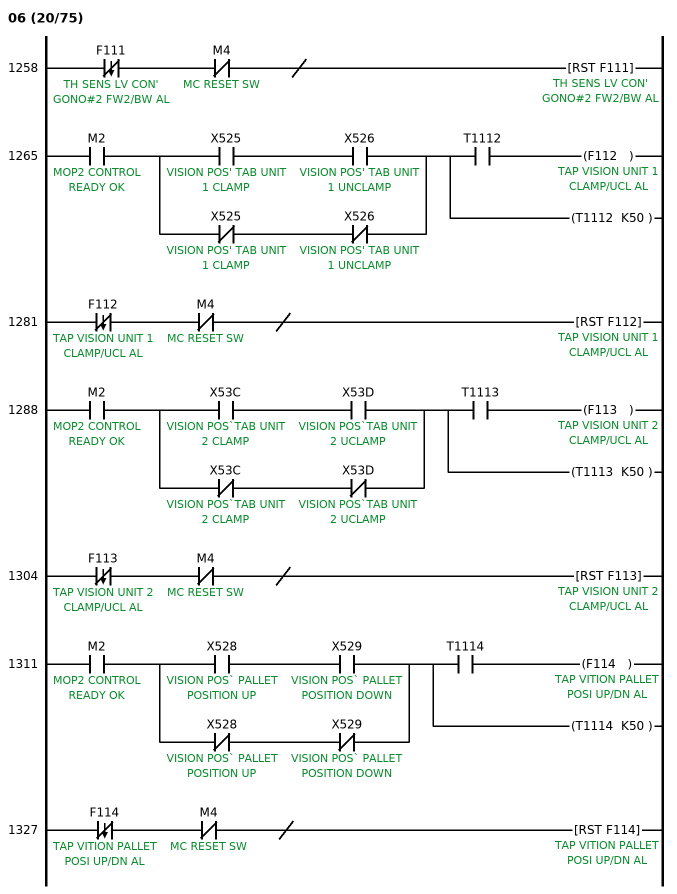
1258  LDFI    F111  ; TH SENS LV CON' GONO#2 FW2/BW AL
      ANI     M4  ; MC RESET SW
      INV
      RST     F111  ; TH SENS LV CON' GONO#2 FW2/BW AL
1265  LD      M2  ; MOP2 CONTROL READY OK
      LD      X525  ; VISION POS' TAB UNIT 1 CLAMP
      AND     X526  ; VISION POS' TAB UNIT 1 UNCLAMP
      LDI     X525  ; VISION POS' TAB UNIT 1 CLAMP
      ANI     X526  ; VISION POS' TAB UNIT 1 UNCLAMP
      ORB
      ANB
      MPS
      AND     T1112
      OUT     F112  ; TAP VISION UNIT 1 CLAMP/UCL AL
      MPP
      OUT     T1112 K50
1281  LDFI    F112  ; TAP VISION UNIT 1 CLAMP/UCL AL
      ANI     M4  ; MC RESET SW
      INV
      RST     F112  ; TAP VISION UNIT 1 CLAMP/UCL AL
1288  LD      M2  ; MOP2 CONTROL READY OK
      LD      X53C  ; VISION POS`TAB UNIT 2 CLAMP
      AND     X53D  ; VISION POS`TAB UNIT 2 UCLAMP
      LDI     X53C  ; VISION POS`TAB UNIT 2 CLAMP
      ANI     X53D  ; VISION POS`TAB UNIT 2 UCLAMP
      ORB
      ANB
      MPS
      AND     T1113
      OUT     F113  ; TAP VISION UNIT 2 CLAMP/UCL AL
      MPP
      OUT     T1113 K50
1304  LDFI    F113  ; TAP VISION UNIT 2 CLAMP/UCL AL
      ANI     M4  ; MC RESET SW
      INV
      RST     F113  ; TAP VISION UNIT 2 CLAMP/UCL AL
1311  LD      M2  ; MOP2 CONTROL READY OK
      LD      X528  ; VISION POS` PALLET POSITION UP
      AND     X529  ; VISION POS` PALLET POSITION DOWN
      LDI     X528  ; VISION POS` PALLET POSITION UP
      ANI     X529  ; VISION POS` PALLET POSITION DOWN
      ORB
      ANB
      MPS
      AND     T1114
      OUT     F114  ; TAP VITION PALLET POSI UP/DN AL
      MPP
      OUT     T1114 K50
1327  LDFI    F114  ; TAP VITION PALLET POSI UP/DN AL
      ANI     M4  ; MC RESET SW
      INV
      RST     F114  ; TAP VITION PALLET POSI UP/DN AL
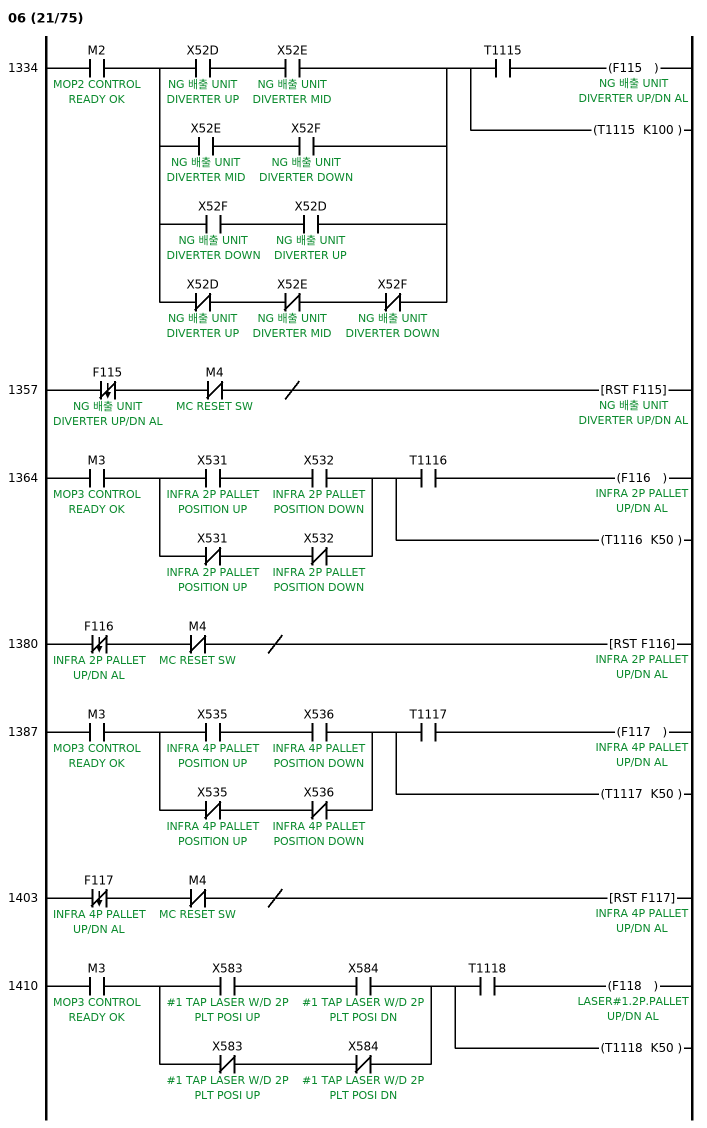
1334  LD      M2  ; MOP2 CONTROL READY OK
      LD      X52D  ; NG 배출 UNIT DIVERTER UP
      AND     X52E  ; NG 배출 UNIT DIVERTER MID
      LD      X52E  ; NG 배출 UNIT DIVERTER MID
      AND     X52F  ; NG 배출 UNIT DIVERTER DOWN
      ORB
      LD      X52F  ; NG 배출 UNIT DIVERTER DOWN
      AND     X52D  ; NG 배출 UNIT DIVERTER UP
      ORB
      LDI     X52D  ; NG 배출 UNIT DIVERTER UP
      ANI     X52E  ; NG 배출 UNIT DIVERTER MID
      ANI     X52F  ; NG 배출 UNIT DIVERTER DOWN
      ORB
      ANB
      MPS
      AND     T1115
      OUT     F115  ; NG 배출 UNIT DIVERTER UP/DN AL
      MPP
      OUT     T1115 K100
1357  LDFI    F115  ; NG 배출 UNIT DIVERTER UP/DN AL
      ANI     M4  ; MC RESET SW
      INV
      RST     F115  ; NG 배출 UNIT DIVERTER UP/DN AL
1364  LD      M3  ; MOP3 CONTROL READY OK
      LD      X531  ; INFRA 2P PALLET POSITION UP
      AND     X532  ; INFRA 2P PALLET POSITION DOWN
      LDI     X531  ; INFRA 2P PALLET POSITION UP
      ANI     X532  ; INFRA 2P PALLET POSITION DOWN
      ORB
      ANB
      MPS
      AND     T1116
      OUT     F116  ; INFRA 2P PALLET UP/DN AL
      MPP
      OUT     T1116 K50
1380  LDFI    F116  ; INFRA 2P PALLET UP/DN AL
      ANI     M4  ; MC RESET SW
      INV
      RST     F116  ; INFRA 2P PALLET UP/DN AL
1387  LD      M3  ; MOP3 CONTROL READY OK
      LD      X535  ; INFRA 4P PALLET POSITION UP
      AND     X536  ; INFRA 4P PALLET POSITION DOWN
      LDI     X535  ; INFRA 4P PALLET POSITION UP
      ANI     X536  ; INFRA 4P PALLET POSITION DOWN
      ORB
      ANB
      MPS
      AND     T1117
      OUT     F117  ; INFRA 4P PALLET UP/DN AL
      MPP
      OUT     T1117 K50
1403  LDFI    F117  ; INFRA 4P PALLET UP/DN AL
      ANI     M4  ; MC RESET SW
      INV
      RST     F117  ; INFRA 4P PALLET UP/DN AL
1410  LD      M3  ; MOP3 CONTROL READY OK
      LD      X583  ; #1 TAP LASER W/D 2P PLT POSI UP
      AND     X584  ; #1 TAP LASER W/D 2P PLT POSI DN
      LDI     X583  ; #1 TAP LASER W/D 2P PLT POSI UP
      ANI     X584  ; #1 TAP LASER W/D 2P PLT POSI DN
      ORB
      ANB
      MPS
      AND     T1118
      OUT     F118  ; LASER#1.2P.PALLET UP/DN AL
      MPP
      OUT     T1118 K50
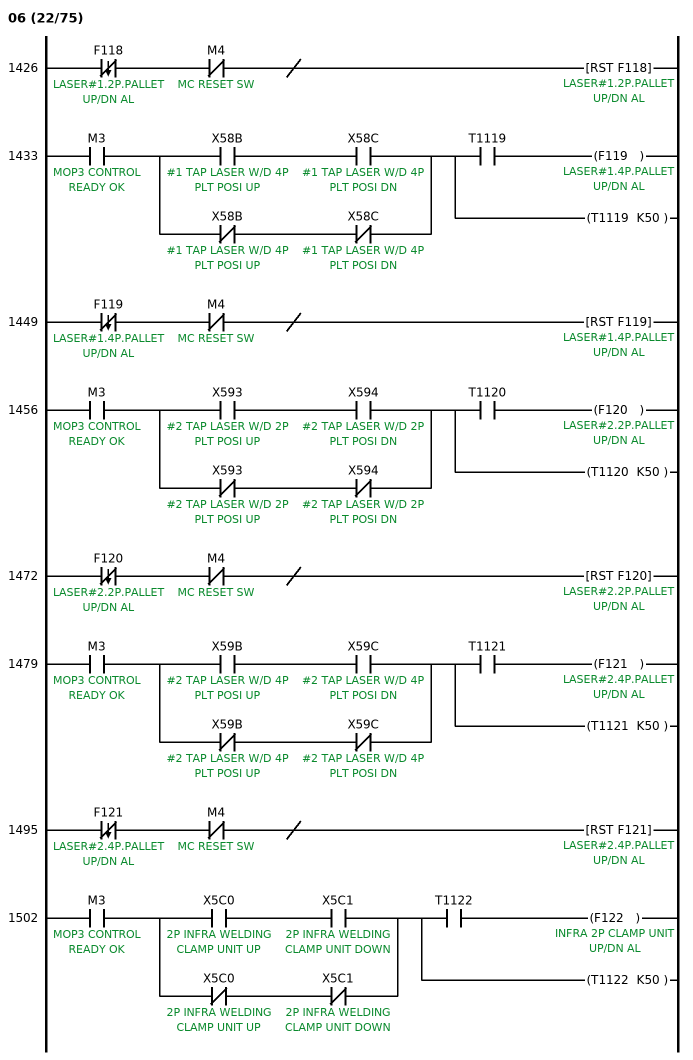
1426  LDFI    F118  ; LASER#1.2P.PALLET UP/DN AL
      ANI     M4  ; MC RESET SW
      INV
      RST     F118  ; LASER#1.2P.PALLET UP/DN AL
1433  LD      M3  ; MOP3 CONTROL READY OK
      LD      X58B  ; #1 TAP LASER W/D 4P PLT POSI UP
      AND     X58C  ; #1 TAP LASER W/D 4P PLT POSI DN
      LDI     X58B  ; #1 TAP LASER W/D 4P PLT POSI UP
      ANI     X58C  ; #1 TAP LASER W/D 4P PLT POSI DN
      ORB
      ANB
      MPS
      AND     T1119
      OUT     F119  ; LASER#1.4P.PALLET UP/DN AL
      MPP
      OUT     T1119 K50
1449  LDFI    F119  ; LASER#1.4P.PALLET UP/DN AL
      ANI     M4  ; MC RESET SW
      INV
      RST     F119  ; LASER#1.4P.PALLET UP/DN AL
1456  LD      M3  ; MOP3 CONTROL READY OK
      LD      X593  ; #2 TAP LASER W/D 2P PLT POSI UP
      AND     X594  ; #2 TAP LASER W/D 2P PLT POSI DN
      LDI     X593  ; #2 TAP LASER W/D 2P PLT POSI UP
      ANI     X594  ; #2 TAP LASER W/D 2P PLT POSI DN
      ORB
      ANB
      MPS
      AND     T1120
      OUT     F120  ; LASER#2.2P.PALLET UP/DN AL
      MPP
      OUT     T1120 K50
1472  LDFI    F120  ; LASER#2.2P.PALLET UP/DN AL
      ANI     M4  ; MC RESET SW
      INV
      RST     F120  ; LASER#2.2P.PALLET UP/DN AL
1479  LD      M3  ; MOP3 CONTROL READY OK
      LD      X59B  ; #2 TAP LASER W/D 4P PLT POSI UP
      AND     X59C  ; #2 TAP LASER W/D 4P PLT POSI DN
      LDI     X59B  ; #2 TAP LASER W/D 4P PLT POSI UP
      ANI     X59C  ; #2 TAP LASER W/D 4P PLT POSI DN
      ORB
      ANB
      MPS
      AND     T1121
      OUT     F121  ; LASER#2.4P.PALLET UP/DN AL
      MPP
      OUT     T1121 K50
1495  LDFI    F121  ; LASER#2.4P.PALLET UP/DN AL
      ANI     M4  ; MC RESET SW
      INV
      RST     F121  ; LASER#2.4P.PALLET UP/DN AL
1502  LD      M3  ; MOP3 CONTROL READY OK
      LD      X5C0  ; 2P INFRA WELDING CLAMP UNIT UP
      AND     X5C1  ; 2P INFRA WELDING CLAMP UNIT DOWN
      LDI     X5C0  ; 2P INFRA WELDING CLAMP UNIT UP
      ANI     X5C1  ; 2P INFRA WELDING CLAMP UNIT DOWN
      ORB
      ANB
      MPS
      AND     T1122
      OUT     F122  ; INFRA 2P CLAMP UNIT UP/DN AL
      MPP
      OUT     T1122 K50
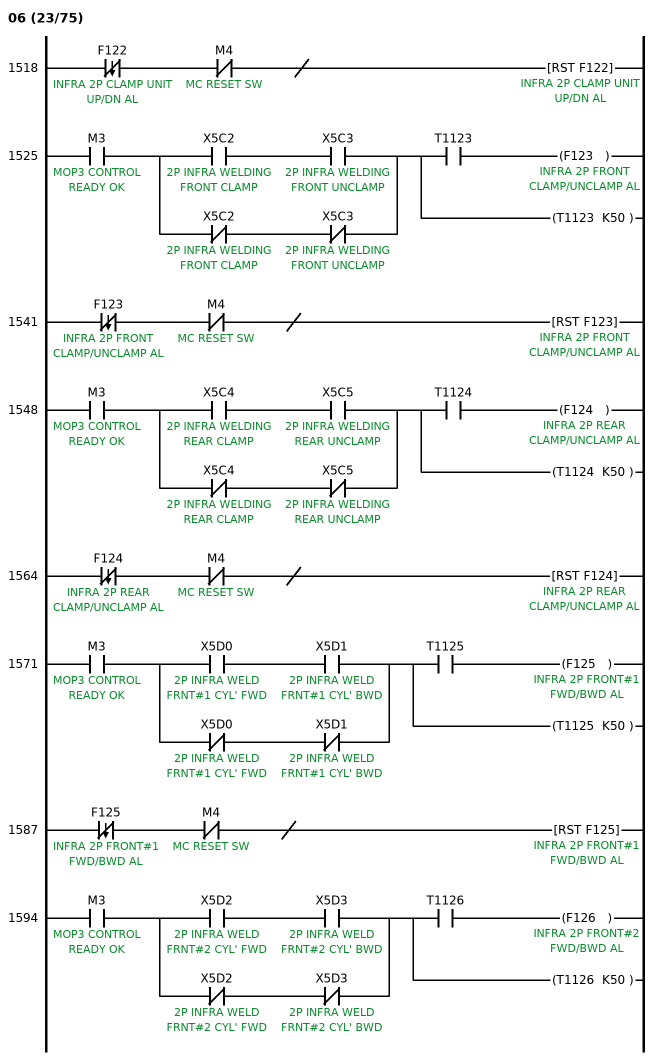
1518  LDFI    F122  ; INFRA 2P CLAMP UNIT UP/DN AL
      ANI     M4  ; MC RESET SW
      INV
      RST     F122  ; INFRA 2P CLAMP UNIT UP/DN AL
1525  LD      M3  ; MOP3 CONTROL READY OK
      LD      X5C2  ; 2P INFRA WELDING FRONT CLAMP
      AND     X5C3  ; 2P INFRA WELDING FRONT UNCLAMP
      LDI     X5C2  ; 2P INFRA WELDING FRONT CLAMP
      ANI     X5C3  ; 2P INFRA WELDING FRONT UNCLAMP
      ORB
      ANB
      MPS
      AND     T1123
      OUT     F123  ; INFRA 2P FRONT CLAMP/UNCLAMP AL
      MPP
      OUT     T1123 K50
1541  LDFI    F123  ; INFRA 2P FRONT CLAMP/UNCLAMP AL
      ANI     M4  ; MC RESET SW
      INV
      RST     F123  ; INFRA 2P FRONT CLAMP/UNCLAMP AL
1548  LD      M3  ; MOP3 CONTROL READY OK
      LD      X5C4  ; 2P INFRA WELDING REAR CLAMP
      AND     X5C5  ; 2P INFRA WELDING REAR UNCLAMP
      LDI     X5C4  ; 2P INFRA WELDING REAR CLAMP
      ANI     X5C5  ; 2P INFRA WELDING REAR UNCLAMP
      ORB
      ANB
      MPS
      AND     T1124
      OUT     F124  ; INFRA 2P REAR CLAMP/UNCLAMP AL
      MPP
      OUT     T1124 K50
1564  LDFI    F124  ; INFRA 2P REAR CLAMP/UNCLAMP AL
      ANI     M4  ; MC RESET SW
      INV
      RST     F124  ; INFRA 2P REAR CLAMP/UNCLAMP AL
1571  LD      M3  ; MOP3 CONTROL READY OK
      LD      X5D0  ; 2P INFRA WELD FRNT#1 CYL' FWD
      AND     X5D1  ; 2P INFRA WELD FRNT#1 CYL' BWD
      LDI     X5D0  ; 2P INFRA WELD FRNT#1 CYL' FWD
      ANI     X5D1  ; 2P INFRA WELD FRNT#1 CYL' BWD
      ORB
      ANB
      MPS
      AND     T1125
      OUT     F125  ; INFRA 2P FRONT#1 FWD/BWD AL
      MPP
      OUT     T1125 K50
1587  LDFI    F125  ; INFRA 2P FRONT#1 FWD/BWD AL
      ANI     M4  ; MC RESET SW
      INV
      RST     F125  ; INFRA 2P FRONT#1 FWD/BWD AL
1594  LD      M3  ; MOP3 CONTROL READY OK
      LD      X5D2  ; 2P INFRA WELD FRNT#2 CYL' FWD
      AND     X5D3  ; 2P INFRA WELD FRNT#2 CYL' BWD
      LDI     X5D2  ; 2P INFRA WELD FRNT#2 CYL' FWD
      ANI     X5D3  ; 2P INFRA WELD FRNT#2 CYL' BWD
      ORB
      ANB
      MPS
      AND     T1126
      OUT     F126  ; INFRA 2P FRONT#2 FWD/BWD AL
      MPP
      OUT     T1126 K50
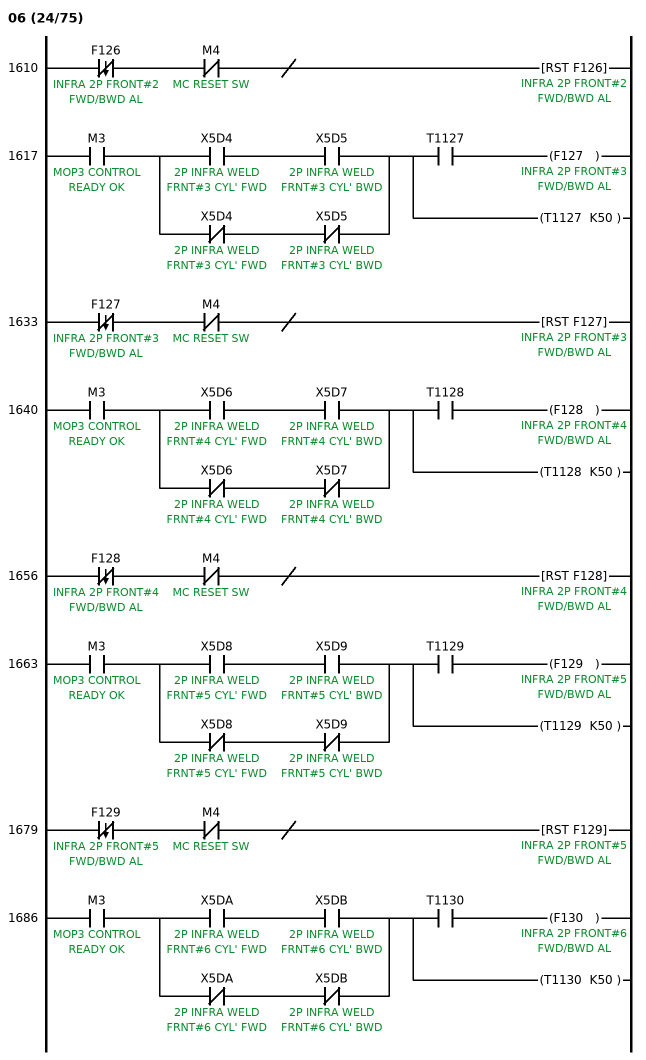
1610  LDFI    F126  ; INFRA 2P FRONT#2 FWD/BWD AL
      ANI     M4  ; MC RESET SW
      INV
      RST     F126  ; INFRA 2P FRONT#2 FWD/BWD AL
1617  LD      M3  ; MOP3 CONTROL READY OK
      LD      X5D4  ; 2P INFRA WELD FRNT#3 CYL' FWD
      AND     X5D5  ; 2P INFRA WELD FRNT#3 CYL' BWD
      LDI     X5D4  ; 2P INFRA WELD FRNT#3 CYL' FWD
      ANI     X5D5  ; 2P INFRA WELD FRNT#3 CYL' BWD
      ORB
      ANB
      MPS
      AND     T1127
      OUT     F127  ; INFRA 2P FRONT#3 FWD/BWD AL
      MPP
      OUT     T1127 K50
1633  LDFI    F127  ; INFRA 2P FRONT#3 FWD/BWD AL
      ANI     M4  ; MC RESET SW
      INV
      RST     F127  ; INFRA 2P FRONT#3 FWD/BWD AL
1640  LD      M3  ; MOP3 CONTROL READY OK
      LD      X5D6  ; 2P INFRA WELD FRNT#4 CYL' FWD
      AND     X5D7  ; 2P INFRA WELD FRNT#4 CYL' BWD
      LDI     X5D6  ; 2P INFRA WELD FRNT#4 CYL' FWD
      ANI     X5D7  ; 2P INFRA WELD FRNT#4 CYL' BWD
      ORB
      ANB
      MPS
      AND     T1128
      OUT     F128  ; INFRA 2P FRONT#4 FWD/BWD AL
      MPP
      OUT     T1128 K50
1656  LDFI    F128  ; INFRA 2P FRONT#4 FWD/BWD AL
      ANI     M4  ; MC RESET SW
      INV
      RST     F128  ; INFRA 2P FRONT#4 FWD/BWD AL
1663  LD      M3  ; MOP3 CONTROL READY OK
      LD      X5D8  ; 2P INFRA WELD FRNT#5 CYL' FWD
      AND     X5D9  ; 2P INFRA WELD FRNT#5 CYL' BWD
      LDI     X5D8  ; 2P INFRA WELD FRNT#5 CYL' FWD
      ANI     X5D9  ; 2P INFRA WELD FRNT#5 CYL' BWD
      ORB
      ANB
      MPS
      AND     T1129
      OUT     F129  ; INFRA 2P FRONT#5 FWD/BWD AL
      MPP
      OUT     T1129 K50
1679  LDFI    F129  ; INFRA 2P FRONT#5 FWD/BWD AL
      ANI     M4  ; MC RESET SW
      INV
      RST     F129  ; INFRA 2P FRONT#5 FWD/BWD AL
1686  LD      M3  ; MOP3 CONTROL READY OK
      LD      X5DA  ; 2P INFRA WELD FRNT#6 CYL' FWD
      AND     X5DB  ; 2P INFRA WELD FRNT#6 CYL' BWD
      LDI     X5DA  ; 2P INFRA WELD FRNT#6 CYL' FWD
      ANI     X5DB  ; 2P INFRA WELD FRNT#6 CYL' BWD
      ORB
      ANB
      MPS
      AND     T1130
      OUT     F130  ; INFRA 2P FRONT#6 FWD/BWD AL
      MPP
      OUT     T1130 K50
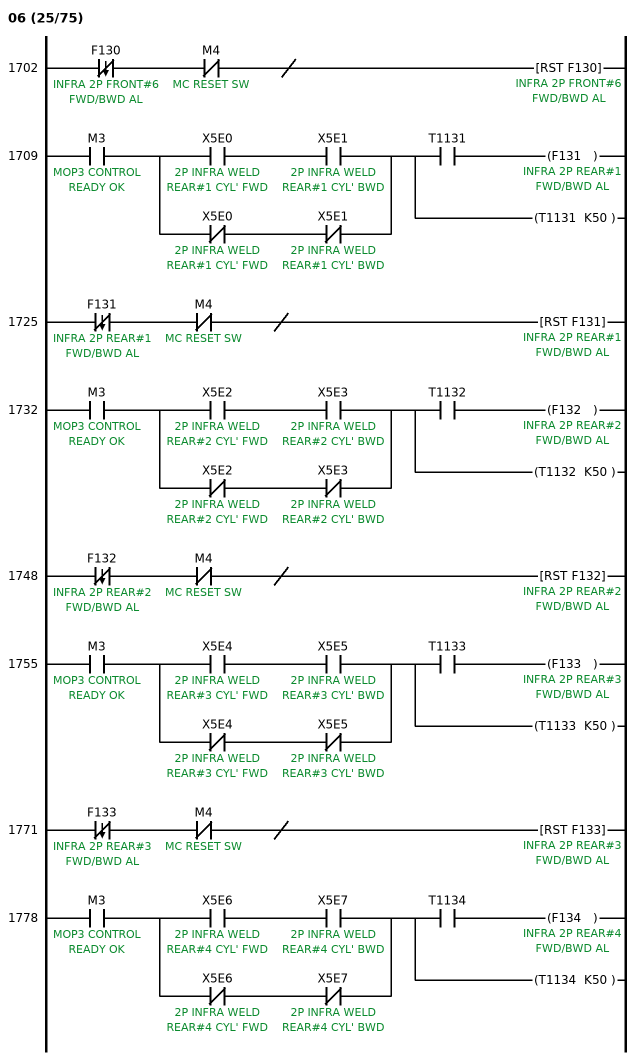
1702  LDFI    F130  ; INFRA 2P FRONT#6 FWD/BWD AL
      ANI     M4  ; MC RESET SW
      INV
      RST     F130  ; INFRA 2P FRONT#6 FWD/BWD AL
1709  LD      M3  ; MOP3 CONTROL READY OK
      LD      X5E0  ; 2P INFRA WELD REAR#1 CYL' FWD
      AND     X5E1  ; 2P INFRA WELD REAR#1 CYL' BWD
      LDI     X5E0  ; 2P INFRA WELD REAR#1 CYL' FWD
      ANI     X5E1  ; 2P INFRA WELD REAR#1 CYL' BWD
      ORB
      ANB
      MPS
      AND     T1131
      OUT     F131  ; INFRA 2P REAR#1 FWD/BWD AL
      MPP
      OUT     T1131 K50
1725  LDFI    F131  ; INFRA 2P REAR#1 FWD/BWD AL
      ANI     M4  ; MC RESET SW
      INV
      RST     F131  ; INFRA 2P REAR#1 FWD/BWD AL
1732  LD      M3  ; MOP3 CONTROL READY OK
      LD      X5E2  ; 2P INFRA WELD REAR#2 CYL' FWD
      AND     X5E3  ; 2P INFRA WELD REAR#2 CYL' BWD
      LDI     X5E2  ; 2P INFRA WELD REAR#2 CYL' FWD
      ANI     X5E3  ; 2P INFRA WELD REAR#2 CYL' BWD
      ORB
      ANB
      MPS
      AND     T1132
      OUT     F132  ; INFRA 2P REAR#2 FWD/BWD AL
      MPP
      OUT     T1132 K50
1748  LDFI    F132  ; INFRA 2P REAR#2 FWD/BWD AL
      ANI     M4  ; MC RESET SW
      INV
      RST     F132  ; INFRA 2P REAR#2 FWD/BWD AL
1755  LD      M3  ; MOP3 CONTROL READY OK
      LD      X5E4  ; 2P INFRA WELD REAR#3 CYL' FWD
      AND     X5E5  ; 2P INFRA WELD REAR#3 CYL' BWD
      LDI     X5E4  ; 2P INFRA WELD REAR#3 CYL' FWD
      ANI     X5E5  ; 2P INFRA WELD REAR#3 CYL' BWD
      ORB
      ANB
      MPS
      AND     T1133
      OUT     F133  ; INFRA 2P REAR#3 FWD/BWD AL
      MPP
      OUT     T1133 K50
1771  LDFI    F133  ; INFRA 2P REAR#3 FWD/BWD AL
      ANI     M4  ; MC RESET SW
      INV
      RST     F133  ; INFRA 2P REAR#3 FWD/BWD AL
1778  LD      M3  ; MOP3 CONTROL READY OK
      LD      X5E6  ; 2P INFRA WELD REAR#4 CYL' FWD
      AND     X5E7  ; 2P INFRA WELD REAR#4 CYL' BWD
      LDI     X5E6  ; 2P INFRA WELD REAR#4 CYL' FWD
      ANI     X5E7  ; 2P INFRA WELD REAR#4 CYL' BWD
      ORB
      ANB
      MPS
      AND     T1134
      OUT     F134  ; INFRA 2P REAR#4 FWD/BWD AL
      MPP
      OUT     T1134 K50
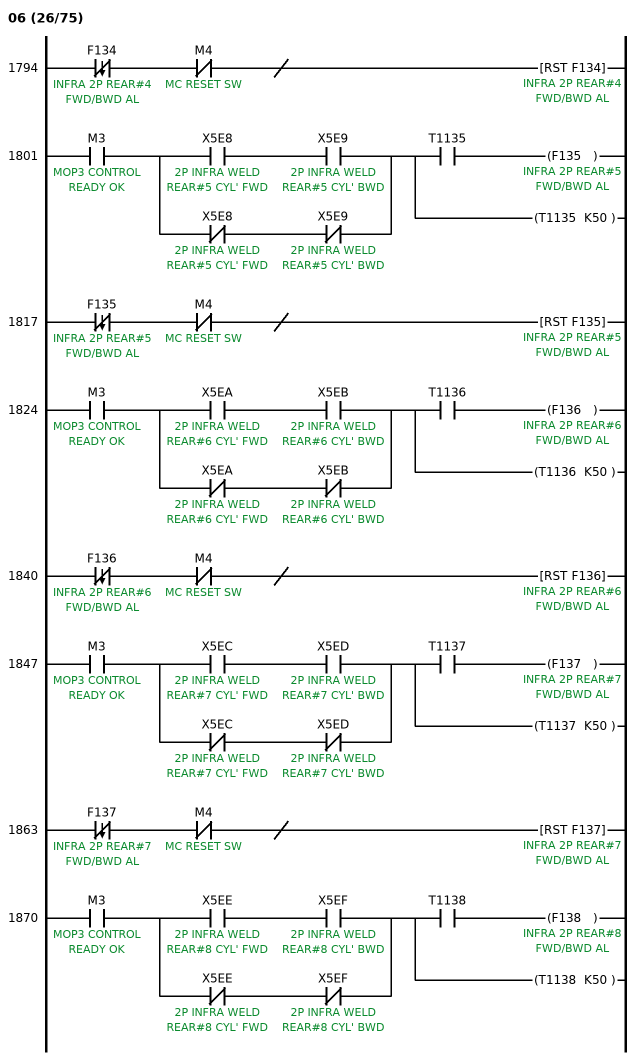
1794  LDFI    F134  ; INFRA 2P REAR#4 FWD/BWD AL
      ANI     M4  ; MC RESET SW
      INV
      RST     F134  ; INFRA 2P REAR#4 FWD/BWD AL
1801  LD      M3  ; MOP3 CONTROL READY OK
      LD      X5E8  ; 2P INFRA WELD REAR#5 CYL' FWD
      AND     X5E9  ; 2P INFRA WELD REAR#5 CYL' BWD
      LDI     X5E8  ; 2P INFRA WELD REAR#5 CYL' FWD
      ANI     X5E9  ; 2P INFRA WELD REAR#5 CYL' BWD
      ORB
      ANB
      MPS
      AND     T1135
      OUT     F135  ; INFRA 2P REAR#5 FWD/BWD AL
      MPP
      OUT     T1135 K50
1817  LDFI    F135  ; INFRA 2P REAR#5 FWD/BWD AL
      ANI     M4  ; MC RESET SW
      INV
      RST     F135  ; INFRA 2P REAR#5 FWD/BWD AL
1824  LD      M3  ; MOP3 CONTROL READY OK
      LD      X5EA  ; 2P INFRA WELD REAR#6 CYL' FWD
      AND     X5EB  ; 2P INFRA WELD REAR#6 CYL' BWD
      LDI     X5EA  ; 2P INFRA WELD REAR#6 CYL' FWD
      ANI     X5EB  ; 2P INFRA WELD REAR#6 CYL' BWD
      ORB
      ANB
      MPS
      AND     T1136
      OUT     F136  ; INFRA 2P REAR#6 FWD/BWD AL
      MPP
      OUT     T1136 K50
1840  LDFI    F136  ; INFRA 2P REAR#6 FWD/BWD AL
      ANI     M4  ; MC RESET SW
      INV
      RST     F136  ; INFRA 2P REAR#6 FWD/BWD AL
1847  LD      M3  ; MOP3 CONTROL READY OK
      LD      X5EC  ; 2P INFRA WELD REAR#7 CYL' FWD
      AND     X5ED  ; 2P INFRA WELD REAR#7 CYL' BWD
      LDI     X5EC  ; 2P INFRA WELD REAR#7 CYL' FWD
      ANI     X5ED  ; 2P INFRA WELD REAR#7 CYL' BWD
      ORB
      ANB
      MPS
      AND     T1137
      OUT     F137  ; INFRA 2P REAR#7 FWD/BWD AL
      MPP
      OUT     T1137 K50
1863  LDFI    F137  ; INFRA 2P REAR#7 FWD/BWD AL
      ANI     M4  ; MC RESET SW
      INV
      RST     F137  ; INFRA 2P REAR#7 FWD/BWD AL
1870  LD      M3  ; MOP3 CONTROL READY OK
      LD      X5EE  ; 2P INFRA WELD REAR#8 CYL' FWD
      AND     X5EF  ; 2P INFRA WELD REAR#8 CYL' BWD
      LDI     X5EE  ; 2P INFRA WELD REAR#8 CYL' FWD
      ANI     X5EF  ; 2P INFRA WELD REAR#8 CYL' BWD
      ORB
      ANB
      MPS
      AND     T1138
      OUT     F138  ; INFRA 2P REAR#8 FWD/BWD AL
      MPP
      OUT     T1138 K50
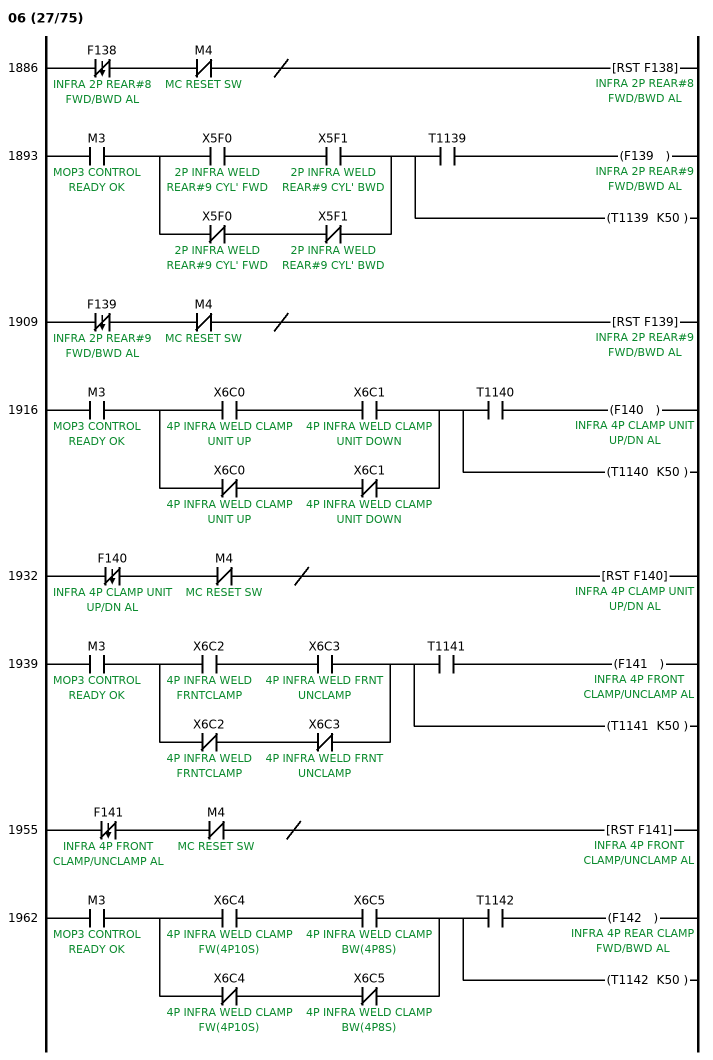
1886  LDFI    F138  ; INFRA 2P REAR#8 FWD/BWD AL
      ANI     M4  ; MC RESET SW
      INV
      RST     F138  ; INFRA 2P REAR#8 FWD/BWD AL
1893  LD      M3  ; MOP3 CONTROL READY OK
      LD      X5F0  ; 2P INFRA WELD REAR#9 CYL' FWD
      AND     X5F1  ; 2P INFRA WELD REAR#9 CYL' BWD
      LDI     X5F0  ; 2P INFRA WELD REAR#9 CYL' FWD
      ANI     X5F1  ; 2P INFRA WELD REAR#9 CYL' BWD
      ORB
      ANB
      MPS
      AND     T1139
      OUT     F139  ; INFRA 2P REAR#9 FWD/BWD AL
      MPP
      OUT     T1139 K50
1909  LDFI    F139  ; INFRA 2P REAR#9 FWD/BWD AL
      ANI     M4  ; MC RESET SW
      INV
      RST     F139  ; INFRA 2P REAR#9 FWD/BWD AL
1916  LD      M3  ; MOP3 CONTROL READY OK
      LD      X6C0  ; 4P INFRA WELD CLAMP UNIT UP
      AND     X6C1  ; 4P INFRA WELD CLAMP UNIT DOWN
      LDI     X6C0  ; 4P INFRA WELD CLAMP UNIT UP
      ANI     X6C1  ; 4P INFRA WELD CLAMP UNIT DOWN
      ORB
      ANB
      MPS
      AND     T1140
      OUT     F140  ; INFRA 4P CLAMP UNIT UP/DN AL
      MPP
      OUT     T1140 K50
1932  LDFI    F140  ; INFRA 4P CLAMP UNIT UP/DN AL
      ANI     M4  ; MC RESET SW
      INV
      RST     F140  ; INFRA 4P CLAMP UNIT UP/DN AL
1939  LD      M3  ; MOP3 CONTROL READY OK
      LD      X6C2  ; 4P INFRA WELD FRNTCLAMP
      AND     X6C3  ; 4P INFRA WELD FRNT UNCLAMP
      LDI     X6C2  ; 4P INFRA WELD FRNTCLAMP
      ANI     X6C3  ; 4P INFRA WELD FRNT UNCLAMP
      ORB
      ANB
      MPS
      AND     T1141
      OUT     F141  ; INFRA 4P FRONT CLAMP/UNCLAMP AL
      MPP
      OUT     T1141 K50
1955  LDFI    F141  ; INFRA 4P FRONT CLAMP/UNCLAMP AL
      ANI     M4  ; MC RESET SW
      INV
      RST     F141  ; INFRA 4P FRONT CLAMP/UNCLAMP AL
1962  LD      M3  ; MOP3 CONTROL READY OK
      LD      X6C4  ; 4P INFRA WELD CLAMP FW(4P10S)
      AND     X6C5  ; 4P INFRA WELD CLAMP BW(4P8S)
      LDI     X6C4  ; 4P INFRA WELD CLAMP FW(4P10S)
      ANI     X6C5  ; 4P INFRA WELD CLAMP BW(4P8S)
      ORB
      ANB
      MPS
      AND     T1142
      OUT     F142  ; INFRA 4P REAR CLAMP FWD/BWD AL
      MPP
      OUT     T1142 K50
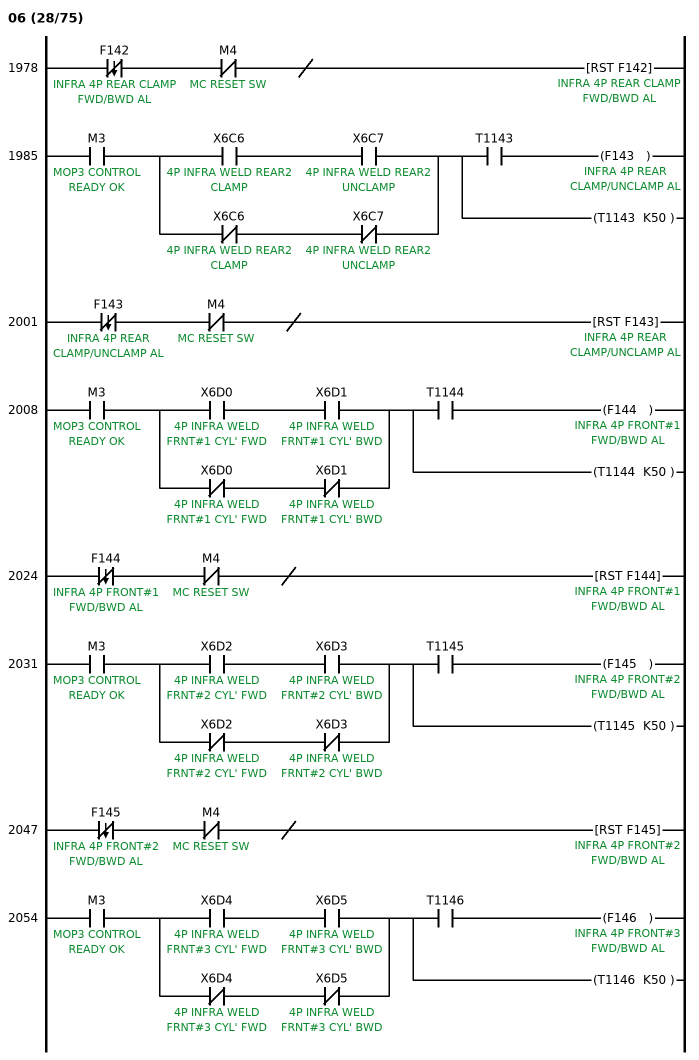
1978  LDFI    F142  ; INFRA 4P REAR CLAMP FWD/BWD AL
      ANI     M4  ; MC RESET SW
      INV
      RST     F142  ; INFRA 4P REAR CLAMP FWD/BWD AL
1985  LD      M3  ; MOP3 CONTROL READY OK
      LD      X6C6  ; 4P INFRA WELD REAR2 CLAMP
      AND     X6C7  ; 4P INFRA WELD REAR2 UNCLAMP
      LDI     X6C6  ; 4P INFRA WELD REAR2 CLAMP
      ANI     X6C7  ; 4P INFRA WELD REAR2 UNCLAMP
      ORB
      ANB
      MPS
      AND     T1143
      OUT     F143  ; INFRA 4P REAR CLAMP/UNCLAMP AL
      MPP
      OUT     T1143 K50
2001  LDFI    F143  ; INFRA 4P REAR CLAMP/UNCLAMP AL
      ANI     M4  ; MC RESET SW
      INV
      RST     F143  ; INFRA 4P REAR CLAMP/UNCLAMP AL
2008  LD      M3  ; MOP3 CONTROL READY OK
      LD      X6D0  ; 4P INFRA WELD FRNT#1 CYL' FWD
      AND     X6D1  ; 4P INFRA WELD FRNT#1 CYL' BWD
      LDI     X6D0  ; 4P INFRA WELD FRNT#1 CYL' FWD
      ANI     X6D1  ; 4P INFRA WELD FRNT#1 CYL' BWD
      ORB
      ANB
      MPS
      AND     T1144
      OUT     F144  ; INFRA 4P FRONT#1 FWD/BWD AL
      MPP
      OUT     T1144 K50
2024  LDFI    F144  ; INFRA 4P FRONT#1 FWD/BWD AL
      ANI     M4  ; MC RESET SW
      INV
      RST     F144  ; INFRA 4P FRONT#1 FWD/BWD AL
2031  LD      M3  ; MOP3 CONTROL READY OK
      LD      X6D2  ; 4P INFRA WELD FRNT#2 CYL' FWD
      AND     X6D3  ; 4P INFRA WELD FRNT#2 CYL' BWD
      LDI     X6D2  ; 4P INFRA WELD FRNT#2 CYL' FWD
      ANI     X6D3  ; 4P INFRA WELD FRNT#2 CYL' BWD
      ORB
      ANB
      MPS
      AND     T1145
      OUT     F145  ; INFRA 4P FRONT#2 FWD/BWD AL
      MPP
      OUT     T1145 K50
2047  LDFI    F145  ; INFRA 4P FRONT#2 FWD/BWD AL
      ANI     M4  ; MC RESET SW
      INV
      RST     F145  ; INFRA 4P FRONT#2 FWD/BWD AL
2054  LD      M3  ; MOP3 CONTROL READY OK
      LD      X6D4  ; 4P INFRA WELD FRNT#3 CYL' FWD
      AND     X6D5  ; 4P INFRA WELD FRNT#3 CYL' BWD
      LDI     X6D4  ; 4P INFRA WELD FRNT#3 CYL' FWD
      ANI     X6D5  ; 4P INFRA WELD FRNT#3 CYL' BWD
      ORB
      ANB
      MPS
      AND     T1146
      OUT     F146  ; INFRA 4P FRONT#3 FWD/BWD AL
      MPP
      OUT     T1146 K50
